(* IEC 61131-3 sources: B-R/Processes/EDT (part 2) *)

(* ---- EDTP2S3A_ACTION.st ---- *)
ACTION P2S3A_ACT:
	//设定时间
	FOR i := 0 TO EDTP2S3_STEP_NUM DO
		IF EDTP2S3A_ST[i] < T#5s THEN
			EDTP2S3A_ST[i] := T#5s;
		END_IF;
		EDTP2S3A_STEP[i].set_time := EDTP2S3A_ST[i];
	END_FOR;

	//流程步骤
	ProcessHandleFC(EDTP2S3A,EDTP2S3A_STEP[0],EDTP2S3_STEP_NUM);

	//object 手自动切换
	IF (EDTP2S3A.status.mode <> 0) AND (NOT EDTP2S3A.auto_mode_edge) THEN
		EDTP2S3A.auto_mode_edge := TRUE;
		EDTP2S3A.manual_mode_edge := FALSE;

		EDTTV0601E.control.auto_operate := TRUE;
		EDTTV0601D.control.auto_operate := TRUE;
		EDTTV0601F.control.auto_operate := TRUE;
		EDTXV0641.control.auto_operate := TRUE;
		EDTR05A.control.auto_operate := TRUE;
	END_IF;

	IF (EDTP2S3A.status.mode = 0) AND (NOT EDTP2S3A.manual_mode_edge) THEN
		EDTP2S3A.manual_mode_edge := TRUE;
		EDTP2S3A.auto_mode_edge := FALSE;

		EDTTV0601E.control.manual_operate := TRUE;
		EDTTV0601D.control.manual_operate := TRUE;
		EDTTV0601F.control.manual_operate := TRUE;
		EDTXV0641.control.manual_operate := TRUE;
		EDTR05A.control.manual_operate := TRUE;
	END_IF;

	//错误信号停机
	EDTP2S3A.input.error_signal := (EDTTV0601E.status.valve_status >= 2) OR (EDTR05A.status.motor_status >= 2) OR
	(EDTTV0601D.status.valve_status >= 2) OR (EDTTV0601F.status.valve_status >= 2) OR (EDTXV0641.status.valve_status >= 2);

	IF EDTP2S3A.status.run_state = 1 THEN
		//步骤执行动作
		CASE EDTP2S3A.status.run_step OF
			0:
				//初始化
				IF NOT EDTP2S3A_STEP[0].done THEN
					EDTTV0601E.control.auto_operate := TRUE;
					EDTTV0601D.control.auto_operate := TRUE;
					EDTTV0601F.control.auto_operate := TRUE;
					EDTXV0641.control.auto_operate := TRUE;
					EDTR05A.control.auto_operate := TRUE;
					EDTP2S3A_STEP[0].done := TRUE;
				END_IF;
			1:
				//人工投料
			2:
				CASE p2_step3_2a OF
					0:
						IF NOT EDTP2S3A_STEP[2].done THEN
							p2_step3_2a := 1;
						END_IF;
					1:
						EDTTV0601F.input.auto_open_signal := TRUE;
						IF EDTTV0601F.input.open_feedback_state THEN
							EDTXV0641.input.auto_open_signal := TRUE;
							p2_step3_2a := 2;
						END_IF;
					2:
						TON_38.PT := DINT_TO_TIME(EDTP2S3_PARA_T1 * 1000);
						TON_38.IN := TRUE;
						IF TON_38.Q THEN
							TON_38.IN := FALSE;
							p2_step3_2a := 3;
						END_IF;
					3:
						EDTTV0601F.input.auto_open_signal := FALSE;
						EDTXV0641.input.auto_open_signal := FALSE;
						IF EDTTV0601F.input.close_feedback_state THEN
							p2_step3_2a := 4;
						END_IF;
					4:
						EDTTV0601E.input.auto_open_signal := TRUE;
						IF EDTTV0601E.input.open_feedback_state THEN
							EDTTV0601D.input.auto_open_signal := TRUE;
							IF EDTTV0601D.input.open_feedback_state THEN
								p2_step3_2a := 5;
							END_IF;
						END_IF;
					5:
						IF EDTTIT0601.status.value >= EDTP2S3_PARA_Temp1 THEN
							p2_step3_2a := 0;
							EDTP2S3A_STEP[2].done := TRUE;
						END_IF;
				END_CASE;
				TON_38();
			3:
				//人工确认釜内回收情况
			4:
				EDTTV0601D.input.auto_open_signal := FALSE;
				IF EDTTV0601D.input.close_feedback_state THEN
					EDTTV0601E.input.auto_open_signal := FALSE;
					IF EDTTV0601E.input.close_feedback_state THEN
						EDTTV0601F.input.auto_open_signal := TRUE;
						IF EDTTV0601F.input.open_feedback_state THEN
							EDTP2S3A_STEP[4].done := TRUE;
						END_IF;
					END_IF;
				END_IF;
			5:
				//人工加料
			6:
				CASE p2_step3_6a OF
					0:
						IF NOT EDTP2S3A_STEP[6].done THEN
							p2_step3_6a := 1;
						END_IF;
					1:
						EDTTV0601F.input.auto_open_signal := TRUE;
						IF EDTTV0601F.input.open_feedback_state THEN
							EDTXV0641.input.auto_open_signal := TRUE;
							p2_step3_6a := 2;
						END_IF;
					2:
						TON_39.PT := DINT_TO_TIME(EDTP2S3_PARA_T1 * 1000);
						TON_39.IN := TRUE;
						IF TON_39.Q THEN
							TON_39.IN := FALSE;
							p2_step3_6a := 3;
						END_IF;
					3:
						EDTTV0601F.input.auto_open_signal := FALSE;
						EDTXV0641.input.auto_open_signal := FALSE;
						IF EDTTV0601F.input.close_feedback_state THEN
							p2_step3_6a := 4;
						END_IF;
					4:
						EDTTV0601E.input.auto_open_signal := TRUE;
						IF EDTTV0601E.input.open_feedback_state THEN
							EDTTV0601D.input.auto_open_signal := TRUE;
							IF EDTTV0601D.input.open_feedback_state THEN
								p2_step3_6a := 5;
							END_IF;
						END_IF;
					5:
						IF EDTTIT0601.status.value >= EDTP2S3_PARA_Temp2 THEN
							p2_step3_6a := 0;
							EDTP2S3A_STEP[6].done := TRUE;
						END_IF;
				END_CASE;
				TON_39();
			7:
				//观察釜内情况
			8:
				EDTTV0601D.input.auto_open_signal := FALSE;
				IF EDTTV0601D.input.close_feedback_state THEN
					EDTTV0601E.input.auto_open_signal := FALSE;
					IF EDTTV0601E.input.close_feedback_state THEN
						EDTTV0601F.input.auto_open_signal := TRUE;
						IF EDTTV0601F.input.open_feedback_state THEN
							EDTP2S3A_STEP[8].done := TRUE;
						END_IF;
					END_IF;
				END_IF;
			9:
				//人工进料
			10:
				TON_10.PT := DINT_TO_TIME(EDTP2S3_PARA_T2 * 60 * 1000);
				TON_10.IN := TRUE;
				IF TON_10.Q THEN
					TON_10.IN := FALSE;
					EDTR05A.input.auto_run_signal := FALSE;
					EDTP2S3A_STEP[10].done := TRUE;
				END_IF;
				TON_10();
		END_CASE;
	END_IF;

	//人工确认步骤可用
	IF (EDTP2S3A.status.run_state) AND (NOT EDTP2S3A_STEP[EDTP2S3A.status.run_step].done AND ((EDTP2S3A.status.run_step = 1) OR (EDTP2S3A.status.run_step = 3) OR (EDTP2S3A.status.run_step = 5) OR (EDTP2S3A.status.run_step = 7) OR
		(EDTP2S3A.status.run_step = 9))) THEN
		EDTP2S3A.status.confirm_enable := TRUE;
	ELSE
		EDTP2S3A.status.confirm_enable := FALSE;
	END_IF;

END_ACTION

(* ---- EDTP2S3B_ACTION.st ---- *)
ACTION P2S3B_ACT:
	//设定时间
	FOR i := 0 TO EDTP2S3_STEP_NUM DO
		IF EDTP2S3B_ST[i] < T#5s THEN
			EDTP2S3B_ST[i] := T#5s;
		END_IF;
		EDTP2S3B_STEP[i].set_time := EDTP2S3B_ST[i];
	END_FOR;

	//流程步骤
	ProcessHandleFC(EDTP2S3B,EDTP2S3B_STEP[0],EDTP2S3_STEP_NUM);

	//object 手自动切换
	IF (EDTP2S3B.status.mode <> 0) AND (NOT EDTP2S3B.auto_mode_edge) THEN
		EDTP2S3B.auto_mode_edge := TRUE;
		EDTP2S3B.manual_mode_edge := FALSE;

		EDTTV0603E.control.auto_operate := TRUE;
		EDTTV0603D.control.auto_operate := TRUE;
		EDTTV0603F.control.auto_operate := TRUE;
		EDTXV0642.control.auto_operate := TRUE;
		EDTR05B.control.auto_operate := TRUE;
	END_IF;

	IF (EDTP2S3B.status.mode = 0) AND (NOT EDTP2S3B.manual_mode_edge) THEN
		EDTP2S3B.manual_mode_edge := TRUE;
		EDTP2S3B.auto_mode_edge := FALSE;

		EDTTV0603E.control.manual_operate := TRUE;
		EDTTV0603D.control.manual_operate := TRUE;
		EDTTV0603F.control.manual_operate := TRUE;
		EDTXV0642.control.manual_operate := TRUE;
		EDTR05B.control.manual_operate := TRUE;
	END_IF;

	//错误信号停机
	EDTP2S3B.input.error_signal := (EDTTV0603E.status.valve_status >= 2) OR (EDTR05B.status.motor_status >= 2) OR
	(EDTTV0603D.status.valve_status >= 2) OR (EDTTV0603F.status.valve_status >= 2) OR (EDTXV0642.status.valve_status >= 2);

	IF EDTP2S3B.status.run_state = 1 THEN
		//步骤执行动作
		CASE EDTP2S3B.status.run_step OF
			0:
				//初始化
				IF NOT EDTP2S3B_STEP[0].done THEN
					EDTTV0603E.control.auto_operate := TRUE;
					EDTTV0603D.control.auto_operate := TRUE;
					EDTTV0603F.control.auto_operate := TRUE;
					EDTXV0642.control.auto_operate := TRUE;
					EDTR05B.control.auto_operate := TRUE;
					EDTP2S3B_STEP[0].done := TRUE;
				END_IF;
			1:
				//人工投料
			2:
				CASE p2_step3_2b OF
					0:
						IF NOT EDTP2S3B_STEP[2].done THEN
							p2_step3_2b := 1;
						END_IF;
					1:
						EDTTV0603F.input.auto_open_signal := TRUE;
						IF EDTTV0603F.input.open_feedback_state THEN
							EDTXV0642.input.auto_open_signal := TRUE;
							p2_step3_2b := 2;
						END_IF;
					2:
						TON_44.PT := DINT_TO_TIME(EDTP2S3_PARA_T1 * 1000);
						TON_44.IN := TRUE;
						IF TON_44.Q THEN
							TON_44.IN := FALSE;
							p2_step3_2b := 3;
						END_IF;
					3:
						EDTTV0603F.input.auto_open_signal := FALSE;
						EDTXV0642.input.auto_open_signal := FALSE;
						IF EDTTV0603F.input.close_feedback_state THEN
							p2_step3_2b := 4;
						END_IF;
					4:
						EDTTV0603E.input.auto_open_signal := TRUE;
						IF EDTTV0603E.input.open_feedback_state THEN
							EDTTV0603D.input.auto_open_signal := TRUE;
							IF EDTTV0603D.input.open_feedback_state THEN
								p2_step3_2b := 5;
							END_IF;
						END_IF;
					5:
						IF EDTTIT0603.status.value >= EDTP2S3_PARA_Temp1 THEN
							p2_step3_2b := 0;
							EDTP2S3B_STEP[2].done := TRUE;
						END_IF;
				END_CASE;
				TON_44();
			3:
				//人工确认釜内回收情况
			4:
				EDTTV0603D.input.auto_open_signal := FALSE;
				IF EDTTV0603D.input.close_feedback_state THEN
					EDTTV0603E.input.auto_open_signal := FALSE;
					IF EDTTV0603E.input.close_feedback_state THEN
						EDTTV0603F.input.auto_open_signal := TRUE;
						IF EDTTV0603F.input.open_feedback_state THEN
							EDTP2S3B_STEP[4].done := TRUE;
						END_IF;
					END_IF;
				END_IF;
			5:
				//人工加料
			6:
				CASE p2_step3_6b OF
					0:
						IF NOT EDTP2S3B_STEP[6].done THEN
							p2_step3_6b := 1;
						END_IF;
					1:
						EDTTV0603F.input.auto_open_signal := TRUE;
						IF EDTTV0603F.input.open_feedback_state THEN
							EDTXV0642.input.auto_open_signal := TRUE;
							p2_step3_6b := 2;
						END_IF;
					2:
						TON_47.PT := DINT_TO_TIME(EDTP2S3_PARA_T1 * 1000);
						TON_47.IN := TRUE;
						IF TON_47.Q THEN
							TON_47.IN := FALSE;
							p2_step3_6b := 3;
						END_IF;
					3:
						EDTTV0603F.input.auto_open_signal := FALSE;
						EDTXV0642.input.auto_open_signal := FALSE;
						IF EDTTV0603F.input.close_feedback_state THEN
							p2_step3_6b := 4;
						END_IF;
					4:
						EDTTV0603E.input.auto_open_signal := TRUE;
						IF EDTTV0603E.input.open_feedback_state THEN
							EDTTV0603D.input.auto_open_signal := TRUE;
							IF EDTTV0603D.input.open_feedback_state THEN
								p2_step3_6b := 5;
							END_IF;
						END_IF;
					5:
						IF EDTTIT0603.status.value >= EDTP2S3_PARA_Temp2 THEN
							p2_step3_6b := 0;
							EDTP2S3B_STEP[6].done := TRUE;
						END_IF;
				END_CASE;
				TON_47();
			7:
				//观察釜内情况
			8:
				EDTTV0603D.input.auto_open_signal := FALSE;
				IF EDTTV0603D.input.close_feedback_state THEN
					EDTTV0603E.input.auto_open_signal := FALSE;
					IF EDTTV0603E.input.close_feedback_state THEN
						EDTTV0603F.input.auto_open_signal := TRUE;
						IF EDTTV0603F.input.open_feedback_state THEN
							EDTP2S3B_STEP[8].done := TRUE;
						END_IF;
					END_IF;
				END_IF;
			9:
				//人工进料
			10:
				TON_48.PT := DINT_TO_TIME(EDTP2S3_PARA_T2 * 60 * 1000);
				TON_48.IN := TRUE;
				IF TON_48.Q THEN
					TON_48.IN := FALSE;
					EDTR05B.input.auto_run_signal := FALSE;
					EDTP2S3B_STEP[10].done := TRUE;
				END_IF;
				TON_48();
		END_CASE;
	END_IF;

	//人工确认步骤可用
	IF (EDTP2S3B.status.run_state) AND (NOT EDTP2S3B_STEP[EDTP2S3B.status.run_step].done AND ((EDTP2S3B.status.run_step = 1) OR (EDTP2S3B.status.run_step = 3) OR (EDTP2S3B.status.run_step = 5) OR (EDTP2S3B.status.run_step = 7) OR
		(EDTP2S3B.status.run_step = 9))) THEN
		EDTP2S3B.status.confirm_enable := TRUE;
	ELSE
		EDTP2S3B.status.confirm_enable := FALSE;
	END_IF;

END_ACTION

(* ---- EDTP2S3C_ACTION.st ---- *)
ACTION P2S3C_ACT:
	//设定时间
	FOR i := 0 TO EDTP2S3_STEP_NUM DO
		IF EDTP2S3C_ST[i] < T#5s THEN
			EDTP2S3C_ST[i] := T#5s;
		END_IF;
		EDTP2S3C_STEP[i].set_time := EDTP2S3C_ST[i];
	END_FOR;

	//流程步骤
	ProcessHandleFC(EDTP2S3C,EDTP2S3C_STEP[0],EDTP2S3_STEP_NUM);

	//object 手自动切换
	IF (EDTP2S3C.status.mode <> 0) AND (NOT EDTP2S3C.auto_mode_edge) THEN
		EDTP2S3C.auto_mode_edge := TRUE;
		EDTP2S3C.manual_mode_edge := FALSE;

		EDTTV0605E.control.auto_operate := TRUE;
		EDTTV0605D.control.auto_operate := TRUE;
		EDTTV0605F.control.auto_operate := TRUE;
		EDTXV0643.control.auto_operate := TRUE;
		EDTR05C.control.auto_operate := TRUE;
	END_IF;

	IF (EDTP2S3C.status.mode = 0) AND (NOT EDTP2S3C.manual_mode_edge) THEN
		EDTP2S3C.manual_mode_edge := TRUE;
		EDTP2S3C.auto_mode_edge := FALSE;

		EDTTV0605E.control.manual_operate := TRUE;
		EDTTV0605D.control.manual_operate := TRUE;
		EDTTV0605F.control.manual_operate := TRUE;
		EDTXV0643.control.manual_operate := TRUE;
		EDTR05C.control.manual_operate := TRUE;
	END_IF;

	//错误信号停机
	EDTP2S3C.input.error_signal := (EDTTV0605E.status.valve_status >= 2) OR (EDTR05C.status.motor_status >= 2) OR
	(EDTTV0605D.status.valve_status >= 2) OR (EDTTV0605F.status.valve_status >= 2) OR (EDTXV0643.status.valve_status >= 2);

	IF EDTP2S3C.status.run_state = 1 THEN
		//步骤执行动作
		CASE EDTP2S3C.status.run_step OF
			0:
				//初始化
				IF NOT EDTP2S3C_STEP[0].done THEN
					EDTTV0605E.control.auto_operate := TRUE;
					EDTTV0605D.control.auto_operate := TRUE;
					EDTTV0605F.control.auto_operate := TRUE;
					EDTXV0643.control.auto_operate := TRUE;
					EDTR05C.control.auto_operate := TRUE;
					EDTP2S3C_STEP[0].done := TRUE;
				END_IF;
			1:
				//人工投料
			2:
				CASE p2_step3_2c OF
					0:
						IF NOT EDTP2S3C_STEP[2].done THEN
							p2_step3_2c := 1;
						END_IF;
					1:
						EDTTV0605F.input.auto_open_signal := TRUE;
						IF EDTTV0605F.input.open_feedback_state THEN
							EDTXV0643.input.auto_open_signal := TRUE;
							p2_step3_2c := 2;
						END_IF;
					2:
						TON_50.PT := DINT_TO_TIME(EDTP2S3_PARA_T1 * 1000);
						TON_50.IN := TRUE;
						IF TON_50.Q THEN
							TON_50.IN := FALSE;
							p2_step3_2c := 3;
						END_IF;
					3:
						EDTTV0605F.input.auto_open_signal := FALSE;
						EDTXV0643.input.auto_open_signal := FALSE;
						IF EDTTV0605F.input.close_feedback_state THEN
							p2_step3_2c := 4;
						END_IF;
					4:
						EDTTV0605E.input.auto_open_signal := TRUE;
						IF EDTTV0605E.input.open_feedback_state THEN
							EDTTV0605D.input.auto_open_signal := TRUE;
							IF EDTTV0605D.input.open_feedback_state THEN
								p2_step3_2c := 5;
							END_IF;
						END_IF;
					5:
						IF EDTTIT0605.status.value >= EDTP2S3_PARA_Temp1 THEN
							p2_step3_2c := 0;
							EDTP2S3C_STEP[2].done := TRUE;
						END_IF;
				END_CASE;
				TON_50();
			3:
				//人工确认釜内回收情况
			4:
				EDTTV0605D.input.auto_open_signal := FALSE;
				IF EDTTV0605D.input.close_feedback_state THEN
					EDTTV0605E.input.auto_open_signal := FALSE;
					IF EDTTV0605E.input.close_feedback_state THEN
						EDTTV0605F.input.auto_open_signal := TRUE;
						IF EDTTV0605F.input.open_feedback_state THEN
							EDTP2S3C_STEP[4].done := TRUE;
						END_IF;
					END_IF;
				END_IF;
			5:
				//人工加料
			6:
				CASE p2_step3_6c OF
					0:
						IF NOT EDTP2S3C_STEP[6].done THEN
							p2_step3_6c := 1;
						END_IF;
					1:
						EDTTV0605F.input.auto_open_signal := TRUE;
						IF EDTTV0605F.input.open_feedback_state THEN
							EDTXV0643.input.auto_open_signal := TRUE;
							p2_step3_6c := 2;
						END_IF;
					2:
						TON_51.PT := DINT_TO_TIME(EDTP2S3_PARA_T1 * 1000);
						TON_51.IN := TRUE;
						IF TON_51.Q THEN
							TON_51.IN := FALSE;
							p2_step3_6c := 3;
						END_IF;
					3:
						EDTTV0605F.input.auto_open_signal := FALSE;
						EDTXV0643.input.auto_open_signal := FALSE;
						IF EDTTV0605F.input.close_feedback_state THEN
							p2_step3_6c := 4;
						END_IF;
					4:
						EDTTV0605E.input.auto_open_signal := TRUE;
						IF EDTTV0605E.input.open_feedback_state THEN
							EDTTV0605D.input.auto_open_signal := TRUE;
							IF EDTTV0605D.input.open_feedback_state THEN
								p2_step3_6c := 5;
							END_IF;
						END_IF;
					5:
						IF EDTTIT0605.status.value >= EDTP2S3_PARA_Temp2 THEN
							p2_step3_6c := 0;
							EDTP2S3C_STEP[6].done := TRUE;
						END_IF;
				END_CASE;
				TON_51();
			7:
				//观察釜内情况
			8:
				EDTTV0605D.input.auto_open_signal := FALSE;
				IF EDTTV0605D.input.close_feedback_state THEN
					EDTTV0605E.input.auto_open_signal := FALSE;
					IF EDTTV0605E.input.close_feedback_state THEN
						EDTTV0605F.input.auto_open_signal := TRUE;
						IF EDTTV0605F.input.open_feedback_state THEN
							EDTP2S3C_STEP[8].done := TRUE;
						END_IF;
					END_IF;
				END_IF;
			9:
				//人工进料
			10:
				TON_53.PT := DINT_TO_TIME(EDTP2S3_PARA_T2 * 60 * 1000);
				TON_53.IN := TRUE;
				IF TON_53.Q THEN
					TON_53.IN := FALSE;
					EDTR05C.input.auto_run_signal := FALSE;
					EDTP2S3C_STEP[10].done := TRUE;
				END_IF;
				TON_53();
		END_CASE;
	END_IF;

	//人工确认步骤可用
	IF (EDTP2S3C.status.run_state) AND (NOT EDTP2S3C_STEP[EDTP2S3C.status.run_step].done AND ((EDTP2S3C.status.run_step = 1) OR (EDTP2S3C.status.run_step = 3) OR (EDTP2S3C.status.run_step = 5) OR (EDTP2S3C.status.run_step = 7) OR
		(EDTP2S3C.status.run_step = 9))) THEN
		EDTP2S3C.status.confirm_enable := TRUE;
	ELSE
		EDTP2S3C.status.confirm_enable := FALSE;
	END_IF;

END_ACTION

(* ---- EDTP2S3D_ACTION.st ---- *)
ACTION P2S3D_ACT:
	//设定时间
	FOR i := 0 TO EDTP2S3_STEP_NUM DO
		IF EDTP2S3D_ST[i] < T#5s THEN
			EDTP2S3D_ST[i] := T#5s;
		END_IF;
		EDTP2S3D_STEP[i].set_time := EDTP2S3D_ST[i];
	END_FOR;

	//流程步骤
	ProcessHandleFC(EDTP2S3D,EDTP2S3D_STEP[0],EDTP2S3_STEP_NUM);

	//object 手自动切换
	IF (EDTP2S3D.status.mode <> 0) AND (NOT EDTP2S3D.auto_mode_edge) THEN
		EDTP2S3D.auto_mode_edge := TRUE;
		EDTP2S3D.manual_mode_edge := FALSE;

		EDTTV0607E.control.auto_operate := TRUE;
		EDTTV0607D.control.auto_operate := TRUE;
		EDTTV0607F.control.auto_operate := TRUE;
		EDTXV0644.control.auto_operate := TRUE;
		EDTR05D.control.auto_operate := TRUE;
	END_IF;

	IF (EDTP2S3D.status.mode = 0) AND (NOT EDTP2S3D.manual_mode_edge) THEN
		EDTP2S3D.manual_mode_edge := TRUE;
		EDTP2S3D.auto_mode_edge := FALSE;

		EDTTV0607E.control.manual_operate := TRUE;
		EDTTV0607D.control.manual_operate := TRUE;
		EDTTV0607F.control.manual_operate := TRUE;
		EDTXV0644.control.manual_operate := TRUE;
		EDTR05D.control.manual_operate := TRUE;
	END_IF;

	//错误信号停机
	EDTP2S3D.input.error_signal := (EDTTV0607E.status.valve_status >= 2) OR (EDTR05D.status.motor_status >= 2) OR
	(EDTTV0607D.status.valve_status >= 2) OR (EDTTV0607F.status.valve_status >= 2) OR (EDTXV0644.status.valve_status >= 2);

	IF EDTP2S3D.status.run_state = 1 THEN
		//步骤执行动作
		CASE EDTP2S3D.status.run_step OF
			0:
				//初始化
				IF NOT EDTP2S3D_STEP[0].done THEN
					EDTTV0607E.control.auto_operate := TRUE;
					EDTTV0607D.control.auto_operate := TRUE;
					EDTTV0607F.control.auto_operate := TRUE;
					EDTXV0644.control.auto_operate := TRUE;
					EDTR05D.control.auto_operate := TRUE;
					EDTP2S3D_STEP[0].done := TRUE;
				END_IF;
			1:
				//人工投料
			2:
				CASE p2_step3_2d OF
					0:
						IF NOT EDTP2S3D_STEP[2].done THEN
							p2_step3_2d := 1;
						END_IF;
					1:
						EDTTV0607F.input.auto_open_signal := TRUE;
						IF EDTTV0607F.input.open_feedback_state THEN
							EDTXV0644.input.auto_open_signal := TRUE;
							p2_step3_2d := 2;
						END_IF;
					2:
						TON_56.PT := DINT_TO_TIME(EDTP2S3_PARA_T1 * 1000);
						TON_56.IN := TRUE;
						IF TON_56.Q THEN
							TON_56.IN := FALSE;
							p2_step3_2d := 3;
						END_IF;
					3:
						EDTTV0607F.input.auto_open_signal := FALSE;
						EDTXV0644.input.auto_open_signal := FALSE;
						IF EDTTV0607F.input.close_feedback_state THEN
							p2_step3_2d := 4;
						END_IF;
					4:
						EDTTV0607E.input.auto_open_signal := TRUE;
						IF EDTTV0607E.input.open_feedback_state THEN
							EDTTV0607D.input.auto_open_signal := TRUE;
							IF EDTTV0607D.input.open_feedback_state THEN
								p2_step3_2d := 5;
							END_IF;
						END_IF;
					5:
						IF EDTTIT0607.status.value >= EDTP2S3_PARA_Temp1 THEN
							p2_step3_2d := 0;
							EDTP2S3D_STEP[2].done := TRUE;
						END_IF;
				END_CASE;
				TON_56();
			3:
				//人工确认釜内回收情况
			4:
				EDTTV0607D.input.auto_open_signal := FALSE;
				IF EDTTV0607D.input.close_feedback_state THEN
					EDTTV0607E.input.auto_open_signal := FALSE;
					IF EDTTV0607E.input.close_feedback_state THEN
						EDTTV0607F.input.auto_open_signal := TRUE;
						IF EDTTV0607F.input.open_feedback_state THEN
							EDTP2S3D_STEP[4].done := TRUE;
						END_IF;
					END_IF;
				END_IF;
			5:
				//人工加料
			6:
				CASE p2_step3_6d OF
					0:
						IF NOT EDTP2S3D_STEP[6].done THEN
							p2_step3_6d := 1;
						END_IF;
					1:
						EDTTV0607F.input.auto_open_signal := TRUE;
						IF EDTTV0607F.input.open_feedback_state THEN
							EDTXV0644.input.auto_open_signal := TRUE;
							p2_step3_6d := 2;
						END_IF;
					2:
						TON_57.PT := DINT_TO_TIME(EDTP2S3_PARA_T1 * 1000);
						TON_57.IN := TRUE;
						IF TON_57.Q THEN
							TON_57.IN := FALSE;
							p2_step3_6d := 3;
						END_IF;
					3:
						EDTTV0607F.input.auto_open_signal := FALSE;
						EDTXV0644.input.auto_open_signal := FALSE;
						IF EDTTV0607F.input.close_feedback_state THEN
							p2_step3_6d := 4;
						END_IF;
					4:
						EDTTV0607E.input.auto_open_signal := TRUE;
						IF EDTTV0607E.input.open_feedback_state THEN
							EDTTV0607D.input.auto_open_signal := TRUE;
							IF EDTTV0607D.input.open_feedback_state THEN
								p2_step3_6d := 5;
							END_IF;
						END_IF;
					5:
						IF EDTTIT0607.status.value >= EDTP2S3_PARA_Temp2 THEN
							p2_step3_6d := 0;
							EDTP2S3D_STEP[6].done := TRUE;
						END_IF;
				END_CASE;
				TON_57();
			7:
				//观察釜内情况
			8:
				EDTTV0607D.input.auto_open_signal := FALSE;
				IF EDTTV0607D.input.close_feedback_state THEN
					EDTTV0607E.input.auto_open_signal := FALSE;
					IF EDTTV0607E.input.close_feedback_state THEN
						EDTTV0607F.input.auto_open_signal := TRUE;
						IF EDTTV0607F.input.open_feedback_state THEN
							EDTP2S3D_STEP[8].done := TRUE;
						END_IF;
					END_IF;
				END_IF;
			9:
				//人工进料
			10:
				TON_59.PT := DINT_TO_TIME(EDTP2S3_PARA_T2 * 60 * 1000);
				TON_59.IN := TRUE;
				IF TON_59.Q THEN
					TON_59.IN := FALSE;
					EDTR05D.input.auto_run_signal := FALSE;
					EDTP2S3D_STEP[10].done := TRUE;
				END_IF;
				TON_59();
		END_CASE;
	END_IF;

	//人工确认步骤可用
	IF (EDTP2S3D.status.run_state) AND (NOT EDTP2S3D_STEP[EDTP2S3D.status.run_step].done AND ((EDTP2S3D.status.run_step = 1) OR (EDTP2S3D.status.run_step = 3) OR (EDTP2S3D.status.run_step = 5) OR (EDTP2S3D.status.run_step = 7) OR
		(EDTP2S3D.status.run_step = 9))) THEN
		EDTP2S3D.status.confirm_enable := TRUE;
	ELSE
		EDTP2S3D.status.confirm_enable := FALSE;
	END_IF;

END_ACTION

(* ---- EDTP2S4A_ACTION.st ---- *)
ACTION P2S4A_ACT:
	//设定时间
	FOR i := 0 TO EDTP2S4_STEP_NUM DO
		IF EDTP2S4A_ST[i] < T#5s THEN
			EDTP2S4A_ST[i] := T#5s;
		END_IF;
		EDTP2S4A_STEP[i].set_time := EDTP2S4A_ST[i];
	END_FOR;

	//流程步骤
	ProcessHandleFC(EDTP2S4A,EDTP2S4A_STEP[0],EDTP2S4_STEP_NUM);

	//object 手自动切换
	IF (EDTP2S4A.status.mode <> 0) AND (NOT EDTP2S4A.auto_mode_edge) THEN
		EDTP2S4A.auto_mode_edge := TRUE;
		EDTP2S4A.manual_mode_edge := FALSE;

		EDTXV0711.control.auto_operate := TRUE;
		EDTAV0701B.control.auto_operate := TRUE;
		EDTAV0701A.control.auto_operate := TRUE;
		EDTXV0701.control.auto_operate := TRUE;
		EDTR12A.control.auto_operate := TRUE;
		EDTTV0701C.control.auto_operate := TRUE;
		EDTTV0701D.control.auto_operate := TRUE;
		EDTTV0701E.control.auto_operate := TRUE;
		EDTTV0701F.control.auto_operate := TRUE;
		EDTFVT0701.control.auto_operate := TRUE;
		EDTXV0704.control.auto_operate := TRUE;
		EDTXV0705.control.auto_operate := TRUE;
		EDTTV0701A.control.auto_operate := TRUE;
		EDTTV0701B.control.auto_operate := TRUE;
		EDTXV0708.control.auto_operate := TRUE;
		EDTXV0709.control.auto_operate := TRUE;
		EDTXV0715.control.auto_operate := TRUE;

	END_IF;

	IF (EDTP2S4A.status.mode = 0) AND (NOT EDTP2S4A.manual_mode_edge) THEN
		EDTP2S4A.manual_mode_edge := TRUE;
		EDTP2S4A.auto_mode_edge := FALSE;

		EDTXV0711.control.manual_operate := TRUE;
		EDTAV0701B.control.manual_operate := TRUE;
		EDTAV0701A.control.manual_operate := TRUE;
		EDTXV0701.control.manual_operate := TRUE;
		EDTR12A.control.manual_operate := TRUE;
		EDTTV0701C.control.manual_operate := TRUE;
		EDTTV0701D.control.manual_operate := TRUE;
		EDTTV0701E.control.manual_operate := TRUE;
		EDTTV0701F.control.manual_operate := TRUE;
		EDTFVT0701.control.manual_operate := TRUE;
		EDTXV0704.control.manual_operate := TRUE;
		EDTXV0705.control.manual_operate := TRUE;
		EDTTV0701A.control.manual_operate := TRUE;
		EDTTV0701B.control.manual_operate := TRUE;
		EDTXV0708.control.manual_operate := TRUE;
		EDTXV0709.control.manual_operate := TRUE;
		EDTXV0715.control.manual_operate := TRUE;
	END_IF;

	//错误信号停机
	EDTP2S4A.input.error_signal := (EDTXV0711.status.valve_status >= 2) OR (EDTAV0701B.status.valve_status >= 2) OR
	(EDTR12A.status.motor_status >= 2) OR (EDTAV0701A.status.valve_status >= 2) OR (EDTXV0701.status.valve_status >= 2) OR
	(EDTTV0701C.status.valve_status >= 2) OR (EDTTV0701D.status.valve_status >= 2) OR (EDTTV0701E.status.valve_status >= 2) OR
	(EDTTV0701F.status.valve_status >= 2) OR (EDTXV0704.status.valve_status >= 2) OR (EDTXV0705.status.valve_status >= 2) OR
	(EDTTV0701A.status.valve_status >= 2) OR (EDTTV0701B.status.valve_status >= 2) OR (EDTXV0708.status.valve_status >= 2) OR
	(EDTXV0709.status.valve_status >= 2);

	IF EDTP2S4A.status.run_state = 1 THEN
		//步骤执行动作
		CASE EDTP2S4A.status.run_step OF
			0:
				//初始化
				IF NOT EDTP2S4A_STEP[0].done THEN
					EDTXV0711.control.auto_operate := TRUE;
					EDTAV0701B.control.auto_operate := TRUE;
					EDTAV0701A.control.auto_operate := TRUE;
					EDTXV0701.control.auto_operate := TRUE;
					EDTR12A.control.auto_operate := TRUE;
					EDTTV0701C.control.auto_operate := TRUE;
					EDTTV0701D.control.auto_operate := TRUE;
					EDTTV0701E.control.auto_operate := TRUE;
					EDTTV0701F.control.auto_operate := TRUE;
					EDTFVT0701.control.auto_operate := TRUE;
					EDTXV0704.control.auto_operate := TRUE;
					EDTXV0705.control.auto_operate := TRUE;
					EDTTV0701A.control.auto_operate := TRUE;
					EDTTV0701B.control.auto_operate := TRUE;
					EDTXV0708.control.auto_operate := TRUE;
					EDTXV0709.control.auto_operate := TRUE;
					EDTXV0715.control.auto_operate := TRUE;
					EDTP2S4A_STEP[0].done := TRUE;
				END_IF;
			1:
				//手动分层，完成后点确认
			2:
				//除前馏
				R12A_process1 := TRUE;
				EDTP2S4A_STEP[2].done := TRUE;
			3:
				IF NOT R12A_process1 THEN
					EDTP2S4A_STEP[3].done := TRUE;
				END_IF;
			4:
				//转移确认V19空
			5:
				TON_66.PT := DINT_TO_TIME(EDTP2S4_PARA_T5 * 60 * 1000);
				EDTXV0708.input.auto_open_signal := TRUE;
				IF EDTXV0708.input.open_feedback_state THEN
					TON_66.IN := TRUE;
				END_IF;
				IF TON_66.Q THEN
					TON_66.IN := FALSE;
					EDTP2S4A_STEP[5].done := TRUE;
				END_IF;
				TON_66();
			6:
				//确认R12A空
			7:
				TON_67.PT := DINT_TO_TIME(EDTP2S4_PARA_T6 * 60 * 1000);
				EDTXV0708.input.auto_open_signal := FALSE;
				IF EDTXV0708.input.close_feedback_state THEN
					EDTXV0711.input.auto_open_signal := TRUE;
					EDTAV0701A.input.auto_open_signal := TRUE;
				END_IF;
				IF EDTXV0711.input.open_feedback_state AND EDTAV0701A.input.open_feedback_state THEN
					TON_67.IN := TRUE;
				END_IF;
				IF TON_67.Q THEN
					TON_67.IN := FALSE;
					EDTP2S4A_STEP[7].done := TRUE;
				END_IF;
				TON_67();
			8:
				//确认R06A空
			9:
				R12A_process := TRUE;
				EDTAV0701A.input.auto_open_signal := FALSE;
				IF EDTAV0701A.input.close_feedback_state THEN
					EDTXV0711.input.auto_open_signal := FALSE;
					IF EDTXV0711.input.close_feedback_state THEN
						EDTXV0709.input.auto_open_signal := TRUE;
						IF EDTXV0709.input.open_feedback_state THEN
							EDTXV0715.input.auto_open_signal := TRUE;
							EDTP2S4A_STEP[9].done := TRUE;
						END_IF;
					END_IF;
				END_IF;
			10:
				//确认转移完毕，AV0701B前手阀开度为三分一
			11:
				EDTXV0709.input.auto_open_signal := FALSE;
				EDTXV0715.input.auto_open_signal := FALSE;
				EDTAV0701B.input.auto_open_signal := TRUE;
				EDTXV0711.input.auto_open_signal := TRUE;
				IF EDTXV0709.input.close_feedback_state AND EDTXV0711.input.open_feedback_state AND EDTAV0701B.input.open_feedback_state THEN
					EDTP2S4A_STEP[11].done := TRUE;
				END_IF;
			12:
				//V06-->V22确认转移完毕
			13:
				EDTAV0701B.input.auto_open_signal := FALSE;
				EDTXV0711.input.auto_open_signal := FALSE;
				IF EDTXV0711.input.close_feedback_state AND EDTAV0701B.input.close_feedback_state THEN
					EDTP2S4A_STEP[13].done := TRUE;
				END_IF;
			14:
				IF NOT R12A_process THEN
					EDTP2S4A_STEP[14].done := TRUE;
				END_IF;
			15:
			//转移
		END_CASE;
	END_IF;

	//除前馏
	IF R12A_process1 THEN
		CASE R12A_process1_step OF
			0:
				MTBasicsPID_8.Enable := FALSE;
				EDTXV0701.input.auto_open_signal := TRUE;
				EDTR12A.input.auto_run_signal := TRUE;
				EDTXV0704.input.auto_open_signal := FALSE;
				EDTXV0705.input.auto_open_signal := FALSE;
				EDTFVT0701.input.auto_degree_set := 0.0;
				IF EDTXV0701.input.open_feedback_state AND EDTR12A.input.run_feedback AND EDTXV0704.input.close_feedback_state AND EDTXV0705.input.close_feedback_state THEN
					R12A_process1_step := 1;
				END_IF;
			1:
				HeatPot_2(ST1 := DINT_TO_TIME(EDTP2S4_PARA_T2 * 1000),
				ST2 := DINT_TO_TIME(EDTP2S4_PARA_T3 * 1000),
				V3 := EDTTV0701C,
				V4 := EDTTV0701D,
				V5 := EDTTV0701E,
				V6 := EDTTV0701F,
				done := R12A_process1_step_1_done);
				IF R12A_process1_step_1_done THEN
					R12A_process1_step_1_done := FALSE;
					R12A_process1_step := 2;
				END_IF;
			2:
				IF EDTTIT0701.status.value >= EDTP2S4_PARA_Temp1 THEN
					EDTTV0701C.input.auto_open_signal := FALSE;
					IF EDTTV0701C.input.close_feedback_state THEN
						R12A_process1_step := 3;
					END_IF;
				END_IF;
			3:
				TON_24.PT := DINT_TO_TIME(EDTP2S4_PARA_T4 * 60 * 1000);
				IF EDTTIT0702.status.value >= EDTP2S4_PARA_Temp4 THEN
					TON_24.IN := TRUE;
				END_IF;
				IF TON_24.Q THEN
					TON_24.IN := FALSE;
					R12A_process1_step := 4;
				END_IF;
			4:
				MTBasicsPID_8.Enable := TRUE;
				EDTXV0705.input.auto_open_signal := FALSE;
				IF EDTXV0705.input.close_feedback_state THEN
					EDTXV0704.input.auto_open_signal := TRUE;
					IF EDTXV0704.input.open_feedback_state THEN
						//EDTFVT0701.input.auto_degree_set := EDTP2S4A_PARA_O1;
						R12A_process1_step := 5;
					END_IF;
				END_IF;
			5:
				TON_24.PT := DINT_TO_TIME(EDTP2S4_PARA_T7 * 1000);
				IF EDTTIT0702.status.value >= EDTP2S4_PARA_Temp2 THEN
					EDTTV0701D.input.auto_open_signal := FALSE;
					IF EDTTV0701D.input.close_feedback_state THEN
						EDTTV0701E.input.auto_open_signal := FALSE;
						EDTTV0701F.input.auto_open_signal := TRUE;
						//IF EDTTV0701E.input.close_feedback_state AND EDTTV0701F.input.open_feedback_state THEN
							TON_24.IN := TRUE;
						//END_IF;
					END_IF;
				END_IF;
				IF TON_24.Q THEN
					TON_24.IN := FALSE;
					R12A_process1_step := 6;
				END_IF;
			6:
				EDTTV0701F.input.auto_open_signal := FALSE;
				IF EDTTV0701F.input.close_feedback_state THEN
					EDTTV0701A.input.auto_open_signal := TRUE;
					IF EDTTV0701A.input.open_feedback_state THEN
						EDTTV0701B.input.auto_open_signal := TRUE;
						R12A_process1_step := 7;
					END_IF;
				END_IF;
			7:
				IF EDTTIT0701.status.value <= EDTP2S4_PARA_Temp3 THEN
					MTBasicsPID_8.Enable := FALSE;
					EDTTV0701B.input.auto_open_signal := FALSE;
					EDTTV0701A.input.auto_open_signal := FALSE;
					EDTR12A.input.auto_run_signal := FALSE;
					EDTXV0701.input.auto_open_signal := FALSE;
					EDTFVT0701.input.auto_degree_set := 100.0;
				END_IF;
				IF EDTTV0701A.input.close_feedback_state AND EDTTV0701B.input.close_feedback_state AND (NOT EDTR12A.input.run_feedback) THEN// AND EDTXV0701.input.close_feedback_state THEN
					R12A_process1 := FALSE;
					R12A_process1_step := 0;
				END_IF;
		END_CASE;
		TON_24();
	END_IF;

	//甲醇水蒸馏
	IF R12A_process THEN
		CASE R12A_process_step OF
			0:
				//甲醇水蒸馏准备
				MTBasicsPID_8.Enable := FALSE;
				EDTXV0704.input.auto_open_signal := FALSE;
				EDTXV0705.input.auto_open_signal := FALSE;
				EDTXV0701.input.auto_open_signal := TRUE;
				EDTR12A.input.auto_run_signal := TRUE;
				EDTFVT0701.input.auto_degree_set := 0.0;
				IF EDTXV0701.input.open_feedback_state AND EDTR12A.input.run_feedback AND EDTXV0704.input.close_feedback_state AND EDTXV0705.input.close_feedback_state THEN
					R12A_process_step := 1;
				END_IF;
			1:
				HeatPot_5(ST1 := DINT_TO_TIME(EDTP2S4_PARA_T2 * 1000),
				ST2 := DINT_TO_TIME(EDTP2S4_PARA_T3 * 1000),
				V3 := EDTTV0701C,
				V4 := EDTTV0701D,
				V5 := EDTTV0701E,
				V6 := EDTTV0701F,
				done := R12A_process_step_1_done);
				IF R12A_process_step_1_done THEN
					R12A_process_step_1_done := FALSE;
					R12A_process_step := 2;
				END_IF;
			2:
				IF EDTTIT0701.status.value >= EDTP2S4_PARA_Temp1 THEN
					EDTTV0701C.input.auto_open_signal := FALSE;
					IF EDTTV0701C.input.close_feedback_state THEN
						R12A_process_step := 3;
					END_IF;
				END_IF;
			3:
				TON_69.PT := DINT_TO_TIME(EDTP2S4_PARA_T4 * 60 * 1000);
				IF EDTTIT0702.status.value >= EDTP2S4_PARA_Temp4 THEN
					TON_69.IN := TRUE;
				END_IF;
				IF TON_69.Q THEN
					TON_69.IN := FALSE;
					R12A_process_step := 4;
				END_IF;
			4:
				MTBasicsPID_8.Enable := TRUE;
				EDTXV0705.input.auto_open_signal := FALSE;
				IF EDTXV0705.input.close_feedback_state THEN
					EDTXV0704.input.auto_open_signal := TRUE;
					IF EDTXV0704.input.open_feedback_state THEN
						//EDTFVT0701.input.auto_degree_set := EDTP2S4A_PARA_O2;
						R12A_process_step := 5;
					END_IF;
				END_IF;
			5:
				IF EDTTIT0702.status.value >= EDTP2S4_PARA_Temp5 THEN
					EDTXV0704.input.auto_open_signal := FALSE;
					IF EDTXV0704.input.close_feedback_state THEN
						EDTXV0705.input.auto_open_signal := TRUE;
						IF EDTXV0705.input.open_feedback_state THEN
							//EDTFVT0701.input.auto_degree_set := EDTP2S4A_PARA_O3;
							R12A_process_step := 6;
						END_IF;
					END_IF;
				END_IF;
			6:
				TON_69.PT := DINT_TO_TIME(EDTP2S4_PARA_T7 * 1000);
				IF EDTTIT0702.status.value >= EDTP2S4_PARA_Temp6 THEN
					EDTTV0701D.input.auto_open_signal := FALSE;
					IF EDTTV0701D.input.close_feedback_state THEN
						EDTTV0701E.input.auto_open_signal := FALSE;
						EDTTV0701F.input.auto_open_signal := TRUE;
						//IF EDTTV0701E.input.close_feedback_state AND EDTTV0701F.input.open_feedback_state THEN
							TON_69.IN := TRUE;
						//END_IF;
					END_IF;
				END_IF;
				IF TON_69.Q THEN
					TON_69.IN := FALSE;
					R12A_process_step := 7;
				END_IF;
			7:
				EDTTV0701F.input.auto_open_signal := FALSE;
				IF EDTTV0701F.input.close_feedback_state THEN
					EDTTV0701A.input.auto_open_signal := TRUE;
					IF EDTTV0701A.input.open_feedback_state THEN
						EDTTV0701B.input.auto_open_signal := TRUE;
						R12A_process_step := 8;
					END_IF;
				END_IF;
			8:
				IF EDTTIT0701.status.value <= EDTP2S4_PARA_Temp7 THEN
					MTBasicsPID_8.Enable := FALSE;
					EDTTV0701B.input.auto_open_signal := FALSE;
					EDTTV0701A.input.auto_open_signal := FALSE;
					EDTR12A.input.auto_run_signal := FALSE;
					EDTXV0701.input.auto_open_signal := FALSE;
					EDTFVT0701.input.auto_degree_set := 100.0;
				END_IF;
				IF EDTTV0701A.input.close_feedback_state AND EDTTV0701B.input.close_feedback_state AND (NOT EDTR12A.input.run_feedback) THEN //AND EDTXV0701.input.close_feedback_state THEN note：关反馈有问题 临时去掉
					R12A_process := FALSE;
					R12A_process_step := 0;
				END_IF;
		END_CASE;
		TON_69();
	END_IF;

	//分层
	IF r06a_separate THEN
		CASE r06a_separate_step OF
			0:
				r06a_als_data_last := r06a_als_data;
				EDTAV0701B.control.auto_operate := TRUE;
				r06a_separate_step := 1;
			1:
				TON_3.PT := T#2s;
				TON_3.IN := TRUE;
				IF TON_3.Q THEN
					TON_3.IN := FALSE;
					r06a_separate_step := 2;
				END_IF;
			2:
				IF r06a_als_data_last = r06a_als_data THEN
					r06a_separate := FALSE;
					r06a_separate_step := 0;
				ELSE
					r06a_separate_step := 3;
				END_IF;
			3:
				EDTAV0701B.input.auto_open_signal := TRUE;
				TON_3.PT := T#30s;
				TON_3.IN := TRUE;
				IF TON_3.Q THEN
					TON_3.IN := FALSE;
					r06a_separate_step := 4;
					r06a_als_data_last := r06a_als_data;
				END_IF;
			4:
				IF ABS(r06a_als_data_last - r06a_als_data) >= r06a_als_data_threshold THEN
					EDTAV0701B.input.auto_open_signal := FALSE;
					r06a_separate := FALSE;
					r06a_separate_step := 0;
				END_IF;
		END_CASE;
		TON_3();
	END_IF;

	R_TRIG_0(CLK := EDTFVT0701.status.auto_mode);
	IF R_TRIG_0.Q THEN
		MTBasicsPID_8.Enable := TRUE;
	END_IF;
	F_TRIG_0(CLK := EDTFVT0701.status.auto_mode);
	IF F_TRIG_0.Q THEN
		MTBasicsPID_8.Enable := FALSE;
	END_IF;
	//FVT0701 pid调节
	//	MTBasicsPID_8.Enable := TRUE;
	MTBasicsPID_8.PIDParameters.Gain := EDTPid0701Para.gain;
	MTBasicsPID_8.PIDParameters.IntegrationTime := EDTPid0701Para.integration_time;
	MTBasicsPID_8.PIDParameters.DerivativeTime := EDTPid0701Para.derivative_time;
	MTBasicsPID_8.MinOut := 0.0;
	MTBasicsPID_8.MaxOut := 100.0;
	MTBasicsPID_8.SetValue := EDTPid0701Para.set_value;
	MTBasicsPID_8.ActValue := EDTFIT0701.flowrate;
	MTBasicsPID_8.Update := EDTPid0701.update;
	MTBasicsPID_8();
	EDTPid0701.out := MTBasicsPID_8.Out;
	IF MTBasicsPID_8.Active THEN
		EDTFVT0701.input.auto_degree_set := MTBasicsPID_8.Out + EDTPid0701Para.min_out;
		//	ELSE
		//		EDTFVT0701.input.auto_degree_set := 0.0;
	END_IF;
	IF MTBasicsPID_8.UpdateDone THEN
		EDTPid0701.update := FALSE;
	END_IF;

	//人工确认步骤可用
	IF (EDTP2S4A.status.run_state) AND (NOT EDTP2S4A_STEP[EDTP2S4A.status.run_step].done AND ((EDTP2S4A.status.run_step = 1) OR (EDTP2S4A.status.run_step = 4)
		OR (EDTP2S4A.status.run_step = 6) OR (EDTP2S4A.status.run_step = 8) OR (EDTP2S4A.status.run_step = 10) OR (EDTP2S4A.status.run_step = 12) OR (EDTP2S4A.status.run_step = 15))) THEN
		EDTP2S4A.status.confirm_enable := TRUE;
	ELSE
		EDTP2S4A.status.confirm_enable := FALSE;
	END_IF;

END_ACTION

(* ---- EDTP2S4B_ACTION.st ---- *)
ACTION P2S4B_ACT:
	//设定时间
	FOR i := 0 TO EDTP2S4_STEP_NUM DO
		IF EDTP2S4B_ST[i] < T#5s THEN
			EDTP2S4B_ST[i] := T#5s;
		END_IF;
		EDTP2S4B_STEP[i].set_time := EDTP2S4B_ST[i];
	END_FOR;

	//流程步骤
	ProcessHandleFC(EDTP2S4B,EDTP2S4B_STEP[0],EDTP2S4_STEP_NUM);

	//object 手自动切换
	IF (EDTP2S4B.status.mode <> 0) AND (NOT EDTP2S4B.auto_mode_edge) THEN
		EDTP2S4B.auto_mode_edge := TRUE;
		EDTP2S4B.manual_mode_edge := FALSE;

		EDTXV0724.control.auto_operate := TRUE;
		EDTAV0702B.control.auto_operate := TRUE;
		EDTAV0702A.control.auto_operate := TRUE;
		EDTXV0716.control.auto_operate := TRUE;
		EDTR12B.control.auto_operate := TRUE;
		EDTTV0703C.control.auto_operate := TRUE;
		EDTTV0703D.control.auto_operate := TRUE;
		EDTTV0703E.control.auto_operate := TRUE;
		EDTTV0703F.control.auto_operate := TRUE;
		EDTFVT0703.control.auto_operate := TRUE;
		EDTXV0719.control.auto_operate := TRUE;
		EDTXV0718.control.auto_operate := TRUE;
		EDTTV0703A.control.auto_operate := TRUE;
		EDTTV0703B.control.auto_operate := TRUE;
		EDTXV0722.control.auto_operate := TRUE;
		EDTXV0723.control.auto_operate := TRUE;
		EDTXV0715.control.auto_operate := TRUE;

	END_IF;

	IF (EDTP2S4B.status.mode = 0) AND (NOT EDTP2S4B.manual_mode_edge) THEN
		EDTP2S4B.manual_mode_edge := TRUE;
		EDTP2S4B.auto_mode_edge := FALSE;

		EDTXV0724.control.manual_operate := TRUE;
		EDTAV0702B.control.manual_operate := TRUE;
		EDTAV0702A.control.manual_operate := TRUE;
		EDTXV0716.control.manual_operate := TRUE;
		EDTR12B.control.manual_operate := TRUE;
		EDTTV0703C.control.manual_operate := TRUE;
		EDTTV0703D.control.manual_operate := TRUE;
		EDTTV0703E.control.manual_operate := TRUE;
		EDTTV0703F.control.manual_operate := TRUE;
		EDTFVT0703.control.manual_operate := TRUE;
		EDTXV0719.control.manual_operate := TRUE;
		EDTXV0718.control.manual_operate := TRUE;
		EDTTV0703A.control.manual_operate := TRUE;
		EDTTV0703B.control.manual_operate := TRUE;
		EDTXV0722.control.manual_operate := TRUE;
		EDTXV0723.control.manual_operate := TRUE;
		EDTXV0715.control.manual_operate := TRUE;
	END_IF;

	//错误信号停机
	EDTP2S4B.input.error_signal := (EDTXV0724.status.valve_status >= 2) OR (EDTAV0702B.status.valve_status >= 2) OR
	(EDTR12B.status.motor_status >= 2) OR (EDTAV0702A.status.valve_status >= 2) OR (EDTXV0716.status.valve_status >= 2) OR
	(EDTTV0703C.status.valve_status >= 2) OR (EDTTV0703D.status.valve_status >= 2) OR (EDTTV0703E.status.valve_status >= 2) OR
	(EDTTV0703F.status.valve_status >= 2) OR (EDTXV0719.status.valve_status >= 2) OR (EDTXV0718.status.valve_status >= 2) OR
	(EDTTV0703A.status.valve_status >= 2) OR (EDTTV0703B.status.valve_status >= 2) OR (EDTXV0722.status.valve_status >= 2) OR
	(EDTXV0723.status.valve_status >= 2);

	IF EDTP2S4B.status.run_state = 1 THEN
		//步骤执行动作
		CASE EDTP2S4B.status.run_step OF
			0:
				//初始化
				IF NOT EDTP2S4B_STEP[0].done THEN
					EDTXV0724.control.auto_operate := TRUE;
					EDTAV0702B.control.auto_operate := TRUE;
					EDTAV0702A.control.auto_operate := TRUE;
					EDTXV0716.control.auto_operate := TRUE;
					EDTR12B.control.auto_operate := TRUE;
					EDTTV0703C.control.auto_operate := TRUE;
					EDTTV0703D.control.auto_operate := TRUE;
					EDTTV0703E.control.auto_operate := TRUE;
					EDTTV0703F.control.auto_operate := TRUE;
					EDTFVT0703.control.auto_operate := TRUE;
					EDTXV0719.control.auto_operate := TRUE;
					EDTXV0718.control.auto_operate := TRUE;
					EDTTV0703A.control.auto_operate := TRUE;
					EDTTV0703B.control.auto_operate := TRUE;
					EDTXV0722.control.auto_operate := TRUE;
					EDTXV0723.control.auto_operate := TRUE;
					EDTXV0715.control.auto_operate := TRUE;
					EDTP2S4B_STEP[0].done := TRUE;
				END_IF;
			1:
				//手动分层，完成后点确认
			2:
				//除前馏
				R12B_process1 := TRUE;
				EDTP2S4B_STEP[2].done := TRUE;
			3:
				IF NOT R12B_process1 THEN
					EDTP2S4B_STEP[3].done := TRUE;
				END_IF;
			4:
				//转移确认V19空
			5:
				TON_70.PT := DINT_TO_TIME(EDTP2S4_PARA_T5 * 60 * 1000);
				EDTXV0722.input.auto_open_signal := TRUE;
				IF EDTXV0722.input.open_feedback_state THEN
					TON_70.IN := TRUE;
				END_IF;
				IF TON_70.Q THEN
					TON_70.IN := FALSE;
					EDTP2S4B_STEP[5].done := TRUE;
				END_IF;
				TON_70();
			6:
				//确认R12空
			7:
				TON_71.PT := DINT_TO_TIME(EDTP2S4_PARA_T6 * 60 * 1000);
				EDTXV0722.input.auto_open_signal := FALSE;
				IF EDTXV0722.input.close_feedback_state THEN
					EDTXV0724.input.auto_open_signal := TRUE;
					EDTAV0702A.input.auto_open_signal := TRUE;
				END_IF;
				IF EDTXV0724.input.open_feedback_state AND EDTAV0702A.input.open_feedback_state THEN
					TON_71.IN := TRUE;
				END_IF;
				IF TON_71.Q THEN
					TON_71.IN := FALSE;
					EDTP2S4B_STEP[7].done := TRUE;
				END_IF;
				TON_71();
			8:
				//确认R06空
			9:
				R12B_process := TRUE;
				EDTAV0702A.input.auto_open_signal := FALSE;
				IF EDTAV0702A.input.close_feedback_state THEN
					EDTXV0724.input.auto_open_signal := FALSE;
					IF EDTXV0724.input.close_feedback_state THEN
						EDTXV0723.input.auto_open_signal := TRUE;
						IF EDTXV0723.input.open_feedback_state THEN
							EDTXV0715.input.auto_open_signal := TRUE;
							EDTP2S4B_STEP[9].done := TRUE;
						END_IF;
					END_IF;
				END_IF;
			10:
				//确认转移完毕
			11:
				EDTXV0723.input.auto_open_signal := FALSE;
				EDTXV0715.input.auto_open_signal := FALSE;
				EDTAV0702B.input.auto_open_signal := TRUE;
				EDTXV0724.input.auto_open_signal := TRUE;
				IF EDTXV0723.input.close_feedback_state AND EDTXV0724.input.open_feedback_state AND EDTAV0702B.input.open_feedback_state THEN
					EDTP2S4B_STEP[11].done := TRUE;
				END_IF;
			12:
				//V06-->V22确认转移完毕
			13:
				EDTAV0702B.input.auto_open_signal := FALSE;
				EDTXV0724.input.auto_open_signal := FALSE;
				IF EDTXV0724.input.close_feedback_state AND EDTAV0702B.input.close_feedback_state THEN
					EDTP2S4B_STEP[13].done := TRUE;
				END_IF;
			14:
				IF NOT R12B_process THEN
					EDTP2S4B_STEP[14].done := TRUE;
				END_IF;
			15:
			//转移
		END_CASE;
	END_IF;

	//除前馏
	IF R12B_process1 THEN
		CASE R12B_process1_step OF
			0:
				MTBasicsPID_9.Enable := FALSE;
				EDTXV0716.input.auto_open_signal := TRUE;
				EDTR12B.input.auto_run_signal := TRUE;
				EDTXV0719.input.auto_open_signal := FALSE;
				EDTXV0718.input.auto_open_signal := FALSE;
				EDTFVT0703.input.auto_degree_set := 0.0;
				IF EDTXV0716.input.open_feedback_state AND EDTR12B.input.run_feedback AND EDTXV0719.input.close_feedback_state AND EDTXV0718.input.close_feedback_state THEN
					R12B_process1_step := 1;
				END_IF;
			1:
				HeatPot_6(ST1 := DINT_TO_TIME(EDTP2S4_PARA_T2 * 1000),
				ST2 := DINT_TO_TIME(EDTP2S4_PARA_T3 * 1000),
				V3 := EDTTV0703C,
				V4 := EDTTV0703D,
				V5 := EDTTV0703E,
				V6 := EDTTV0703F,
				done := R12B_process1_step_1_done);
				IF R12B_process1_step_1_done THEN
					R12B_process1_step_1_done := FALSE;
					R12B_process1_step := 2;
				END_IF;
			2:
				IF EDTTIT0703.status.value >= EDTP2S4_PARA_Temp1 THEN
					EDTTV0703C.input.auto_open_signal := FALSE;
					IF EDTTV0703C.input.close_feedback_state THEN
						R12B_process1_step := 3;
					END_IF;
				END_IF;
			3:
				TON_72.PT := DINT_TO_TIME(EDTP2S4_PARA_T4 * 60 * 1000);
				IF EDTTIT0704.status.value >= EDTP2S4_PARA_Temp4 THEN
					TON_72.IN := TRUE;
				END_IF;
				IF TON_72.Q THEN
					TON_72.IN := FALSE;
					R12B_process1_step := 4;
				END_IF;
			4:
				MTBasicsPID_9.Enable := TRUE;
				EDTXV0718.input.auto_open_signal := FALSE;
				IF EDTXV0718.input.close_feedback_state THEN
					EDTXV0719.input.auto_open_signal := TRUE;
					IF EDTXV0719.input.open_feedback_state THEN
						//EDTFVT0703.input.auto_degree_set := EDTP2S4B_PARA_O1;
						R12B_process1_step := 5;
					END_IF;
				END_IF;
			5:
				TON_72.PT := DINT_TO_TIME(EDTP2S4_PARA_T7 * 1000);
				IF EDTTIT0704.status.value >= EDTP2S4_PARA_Temp2 THEN
					EDTTV0703D.input.auto_open_signal := FALSE;
					IF EDTTV0703D.input.close_feedback_state THEN
						EDTTV0703E.input.auto_open_signal := FALSE;
						EDTTV0703F.input.auto_open_signal := TRUE;
						//IF EDTTV0703E.input.close_feedback_state AND EDTTV0703F.input.open_feedback_state THEN
							TON_72.IN := TRUE;
						//END_IF;
					END_IF;
				END_IF;
				IF TON_72.Q THEN
					TON_72.IN := FALSE;
					R12B_process1_step := 6;
				END_IF;
			6:
				EDTTV0703F.input.auto_open_signal := FALSE;
				IF EDTTV0703F.input.close_feedback_state THEN
					EDTTV0703A.input.auto_open_signal := TRUE;
					IF EDTTV0703A.input.open_feedback_state THEN
						EDTTV0703B.input.auto_open_signal := TRUE;
						R12B_process1_step := 7;
					END_IF;
				END_IF;
			7:
				IF EDTTIT0703.status.value <= EDTP2S4_PARA_Temp3 THEN
					MTBasicsPID_9.Enable := FALSE;
					EDTTV0703B.input.auto_open_signal := FALSE;
					EDTTV0703A.input.auto_open_signal := FALSE;
					EDTR12B.input.auto_run_signal := FALSE;
					EDTXV0716.input.auto_open_signal := FALSE;
					EDTFVT0703.input.auto_degree_set := 100.0;
				END_IF;
				IF EDTTV0703A.input.close_feedback_state AND EDTTV0703B.input.close_feedback_state AND (NOT EDTR12B.input.run_feedback) AND EDTXV0716.input.close_feedback_state THEN
					R12B_process1 := FALSE;
					R12B_process1_step := 0;
				END_IF;
		END_CASE;
		TON_72();
	END_IF;

	//甲醇水蒸馏
	IF R12B_process THEN
		CASE R12B_process_step OF
			0:
				//甲醇水蒸馏准备
				MTBasicsPID_9.Enable := FALSE;
				EDTXV0719.input.auto_open_signal := FALSE;
				EDTXV0718.input.auto_open_signal := FALSE;
				EDTXV0716.input.auto_open_signal := TRUE;
				EDTR12B.input.auto_run_signal := TRUE;
				EDTFVT0703.input.auto_degree_set := 0.0;
				IF EDTXV0716.input.open_feedback_state AND EDTR12B.input.run_feedback AND EDTXV0719.input.close_feedback_state AND EDTXV0718.input.close_feedback_state THEN
					R12B_process_step := 1;
				END_IF;
			1:
				HeatPot_10(ST1 := DINT_TO_TIME(EDTP2S4_PARA_T2 * 1000),
				ST2 := DINT_TO_TIME(EDTP2S4_PARA_T3 * 1000),
				V3 := EDTTV0703C,
				V4 := EDTTV0703D,
				V5 := EDTTV0703E,
				V6 := EDTTV0703F,
				done := R12B_process_step_1_done);
				IF R12B_process_step_1_done THEN
					R12B_process_step_1_done := FALSE;
					R12B_process_step := 2;
				END_IF;
			2:
				IF EDTTIT0703.status.value >= EDTP2S4_PARA_Temp1 THEN
					EDTTV0703C.input.auto_open_signal := FALSE;
					IF EDTTV0703C.input.close_feedback_state THEN
						R12B_process_step := 3;
					END_IF;
				END_IF;
			3:
				TON_75.PT := DINT_TO_TIME(EDTP2S4_PARA_T4 * 60 * 1000);
				IF EDTTIT0704.status.value >= EDTP2S4_PARA_Temp4 THEN
					TON_75.IN := TRUE;
				END_IF;
				IF TON_75.Q THEN
					TON_75.IN := FALSE;
					R12B_process_step := 4;
				END_IF;
			4:
				MTBasicsPID_9.Enable := TRUE;
				EDTXV0718.input.auto_open_signal := FALSE;
				IF EDTXV0718.input.close_feedback_state THEN
					EDTXV0719.input.auto_open_signal := TRUE;
					IF EDTXV0719.input.open_feedback_state THEN
						//EDTFVT0703.input.auto_degree_set := EDTP2S4B_PARA_O2;
						R12B_process_step := 5;
					END_IF;
				END_IF;
			5:
				IF EDTTIT0704.status.value >= EDTP2S4_PARA_Temp5 THEN
					EDTXV0719.input.auto_open_signal := FALSE;
					IF EDTXV0719.input.close_feedback_state THEN
						EDTXV0718.input.auto_open_signal := TRUE;
						IF EDTXV0718.input.open_feedback_state THEN
							//EDTFVT0703.input.auto_degree_set := EDTP2S4B_PARA_O3;
							R12B_process_step := 6;
						END_IF;
					END_IF;
				END_IF;
			6:
				TON_75.PT := DINT_TO_TIME(EDTP2S4_PARA_T7 * 1000);
				IF EDTTIT0704.status.value >= EDTP2S4_PARA_Temp6 THEN
					EDTTV0703D.input.auto_open_signal := FALSE;
					IF EDTTV0703D.input.close_feedback_state THEN
						EDTTV0703E.input.auto_open_signal := FALSE;
						EDTTV0703F.input.auto_open_signal := TRUE;
						//IF EDTTV0703E.input.close_feedback_state AND EDTTV0703F.input.open_feedback_state THEN
							TON_75.IN := TRUE;
						//END_IF;
					END_IF;
				END_IF;
				IF TON_75.Q THEN
					TON_75.IN := FALSE;
					R12B_process_step := 7;
				END_IF;
			7:
				EDTTV0703F.input.auto_open_signal := FALSE;
				IF EDTTV0703F.input.close_feedback_state THEN
					EDTTV0703A.input.auto_open_signal := TRUE;
					IF EDTTV0703A.input.open_feedback_state THEN
						EDTTV0703B.input.auto_open_signal := TRUE;
						R12B_process_step := 8;
					END_IF;
				END_IF;
			8:
				IF EDTTIT0703.status.value <= EDTP2S4_PARA_Temp7 THEN
					MTBasicsPID_9.Enable := FALSE;
					EDTTV0703B.input.auto_open_signal := FALSE;
					EDTTV0703A.input.auto_open_signal := FALSE;
					EDTR12B.input.auto_run_signal := FALSE;
					EDTXV0716.input.auto_open_signal := FALSE;
					EDTFVT0703.input.auto_degree_set := 100.0;
				END_IF;
				IF EDTTV0703A.input.close_feedback_state AND EDTTV0703B.input.close_feedback_state AND (NOT EDTR12B.input.run_feedback) AND EDTXV0716.input.close_feedback_state THEN
					R12B_process := FALSE;
					R12B_process_step := 0;
				END_IF;
		END_CASE;
		TON_75();
	END_IF;

	R_TRIG_1(CLK := EDTFVT0703.status.auto_mode);
	IF R_TRIG_1.Q THEN
		MTBasicsPID_9.Enable := TRUE;
	END_IF;
	F_TRIG_1(CLK := EDTFVT0703.status.auto_mode);
	IF F_TRIG_1.Q THEN
		MTBasicsPID_9.Enable := FALSE;
	END_IF;
	//FVT0703 pid调节
	//	MTBasicsPID_9.Enable := TRUE;
	MTBasicsPID_9.PIDParameters.Gain := EDTPid0703Para.gain;
	MTBasicsPID_9.PIDParameters.IntegrationTime := EDTPid0703Para.integration_time;
	MTBasicsPID_9.PIDParameters.DerivativeTime := EDTPid0703Para.derivative_time;
	MTBasicsPID_9.MinOut := 0.0;
	MTBasicsPID_9.MaxOut := 100.0;
	MTBasicsPID_9.SetValue := EDTPid0703Para.set_value;
	MTBasicsPID_9.ActValue := EDTFIT0703.flowrate;
	MTBasicsPID_9.Update := EDTPid0703.update;
	MTBasicsPID_9();
	EDTPid0703.out := MTBasicsPID_9.Out;
	IF MTBasicsPID_9.Active THEN
		EDTFVT0703.input.auto_degree_set := MTBasicsPID_9.Out + EDTPid0703Para.min_out;
		//	ELSE
		//		EDTFVT0703.input.auto_degree_set := 0.0;
	END_IF;
	IF MTBasicsPID_9.UpdateDone THEN
		EDTPid0703.update := FALSE;
	END_IF;

	//人工确认步骤可用
	IF (EDTP2S4B.status.run_state) AND (NOT EDTP2S4B_STEP[EDTP2S4B.status.run_step].done AND ((EDTP2S4B.status.run_step = 1) OR (EDTP2S4B.status.run_step = 4)
		OR (EDTP2S4B.status.run_step = 6) OR (EDTP2S4B.status.run_step = 8) OR (EDTP2S4B.status.run_step = 10) OR (EDTP2S4B.status.run_step = 12) OR (EDTP2S4B.status.run_step = 15))) THEN
		EDTP2S4B.status.confirm_enable := TRUE;
	ELSE
		EDTP2S4B.status.confirm_enable := FALSE;
	END_IF;

END_ACTION

(* ---- EDTP3S1A_ACTION.st ---- *)
ACTION P3S1A_ACT:
	//设定时间
	FOR i := 0 TO EDTP3S1_STEP_NUM DO
		IF EDTP3S1A_ST[i] < T#5s THEN
			EDTP3S1A_ST[i] := T#5s;
		END_IF;
		EDTP3S1A_STEP[i].set_time := EDTP3S1A_ST[i];
	END_FOR;

	//流程步骤
	ProcessHandleFC(EDTP3S1A,EDTP3S1A_STEP[0],EDTP3S1_STEP_NUM);

	//object 手自动切换
	IF (EDTP3S1A.status.mode <> 0) AND (NOT EDTP3S1A.auto_mode_edge) THEN
		EDTP3S1A.auto_mode_edge := TRUE;
		EDTP3S1A.manual_mode_edge := FALSE;

		EDTR18A.control.auto_operate := TRUE;
		EDTTV0801C.control.auto_operate := TRUE;
		EDTTV0801E.control.auto_operate := TRUE;
		EDTTV0801D.control.auto_operate := TRUE;
		EDTTV0801B.control.auto_operate := TRUE;
		EDTTV0801A.control.auto_operate := TRUE;
		EDTXV0812.control.auto_operate := TRUE;
		EDTTVT0801.control.auto_operate := TRUE;
		EDTXV0817.control.auto_operate := TRUE;
		EDTXV2107.control.auto_operate := TRUE;
		EDTXV2113.control.auto_operate := TRUE;
		EDTXV2109.control.auto_operate := TRUE;
	END_IF;

	IF (EDTP3S1A.status.mode = 0) AND (NOT EDTP3S1A.manual_mode_edge) THEN
		EDTP3S1A.manual_mode_edge := TRUE;
		EDTP3S1A.auto_mode_edge := FALSE;

		EDTR18A.control.manual_operate := TRUE;
		EDTTV0801C.control.manual_operate := TRUE;
		EDTTV0801E.control.manual_operate := TRUE;
		EDTTV0801D.control.manual_operate := TRUE;
		EDTTV0801B.control.manual_operate := TRUE;
		EDTTV0801A.control.manual_operate := TRUE;
		EDTXV0812.control.manual_operate := TRUE;
		EDTTVT0801.control.manual_operate := TRUE;
		EDTXV0817.control.manual_operate := TRUE;
		EDTXV2107.control.manual_operate := TRUE;
		EDTXV2113.control.manual_operate := TRUE;
		EDTXV2109.control.manual_operate := TRUE;
	END_IF;

	//错误信号停机
	EDTP3S1A.input.error_signal := (EDTR18A.status.motor_status >= 2) OR (EDTTV0801C.status.valve_status >= 2) OR (EDTTV0801E.status.valve_status >= 2) OR
	(EDTTV0801D.status.valve_status >= 2) OR(EDTTV0801B.status.valve_status >= 2) OR (EDTTV0801A.status.valve_status >= 2) OR (EDTXV0812.status.valve_status >= 2);

	IF EDTP3S1A.status.run_state = 1 THEN
		CASE EDTP3S1A.status.run_step OF
			0:
				IF NOT EDTP3S1A_STEP[0].done THEN
					EDTR18A.control.auto_operate := TRUE;
					EDTTV0801C.control.auto_operate := TRUE;
					EDTTV0801E.control.auto_operate := TRUE;
					EDTTV0801D.control.auto_operate := TRUE;
					EDTTV0801B.control.auto_operate := TRUE;
					EDTTV0801A.control.auto_operate := TRUE;
					EDTXV0812.control.auto_operate := TRUE;
					EDTTVT0801.control.auto_operate := TRUE;
					EDTXV0817.control.auto_operate := TRUE;
					EDTXV2107.control.auto_operate := TRUE;
					EDTXV2113.control.auto_operate := TRUE;
					EDTXV2109.control.auto_operate := TRUE;
					IF EDTXV0801.input.close_feedback_state AND EDTXV0806.input.close_feedback_state AND EDTXV0804.input.close_feedback_state AND EDTFQV0801.input.close_feedback_state
						AND EDTXV0814.input.close_feedback_state AND EDTXV0822.input.close_feedback_state AND EDTXV0817.input.close_feedback_state THEN
						EDTP3S1A_STEP[0].done := TRUE;
					END_IF;
				END_IF;
			1:
				//醚化
				CASE p3_step1_1a OF
					0:
						IF NOT EDTP3S1A_STEP[1].done THEN
							p3_step1_1a := 1;
						END_IF;
					1:
						TON_0.IN := FALSE;
						TON_46.IN := FALSE;
						temp_decrease := FALSE;
						FOR i := 0 TO 50 DO
							EDTTIT0801_avg_record[i] := 0;
						END_FOR;
						EDTTIT0801_avg := 0;
						n := 0;
						temp_offset := 0;
						offset := 0;
						EDTPIT0803_record[0] := REAL_TO_INT(EDTPIT0803_PARA.upper_range * 100);
						EDTPIT0803_record[1] := REAL_TO_INT(EDTPIT0803_PARA.upper_range * 100);
						EDTPIT0803_record[2] := REAL_TO_INT(EDTPIT0803_PARA.upper_range * 100);
						EDTTIT0801_record[0] := REAL_TO_INT(EDTTIT0801_PARA.upper_range * 100);
						EDTTIT0801_record[1] := REAL_TO_INT(EDTTIT0801_PARA.upper_range * 100);
						EDTTIT0801_record[2] := REAL_TO_INT(EDTTIT0801_PARA.upper_range * 100);
						EDTR18A.input.auto_run_signal := TRUE;
						IF EDTR18A.input.run_feedback THEN
							p3_step1_1a := 2;
						END_IF;
					2:
						TON_0.PT := DINT_TO_TIME(EDTP3S1_PARA_T2 * 1000);
						EDTTV0801E.input.auto_open_signal := TRUE;
						IF EDTTV0801E.input.open_feedback_state THEN
							EDTXV0812.input.auto_open_signal := TRUE;
							TON_0.IN := TRUE;
						END_IF;
						IF TON_0.Q THEN
							TON_0.IN := FALSE;
							p3_step1_1a := 3;
						END_IF;
					3:
						//每两秒采集一个数据，连续采集3个，连续下降则判定值开始下降
						TON_0.PT := DINT_TO_TIME(EDTP3S1_PARA_T1 * 1000);
						TON_0.IN := TRUE;
						IF TON_0.Q THEN
							TON_0.IN := FALSE;
							EDTPIT0803_record[offset] := REAL_TO_INT(EDTPIT0803.status.value * 100);
							offset := offset + 1;
						END_IF;
						IF offset > 2 THEN
							offset := 0;
						END_IF;
						IF (EDTPIT0803_record[0] > EDTPIT0803_record[1]) AND (EDTPIT0803_record[1] > EDTPIT0803_record[2]) THEN
							p3_step1_1a := 4;
						END_IF;
					4:
						IF EDTPIT0803.status.value <= EDTP3S1_PARA_P3 THEN
							EDTXV0812.input.auto_open_signal := FALSE;
						END_IF;
						IF EDTPIT0803.status.value <= EDTP3S1_PARA_P4 THEN
							EDTTV0801E.input.auto_open_signal := FALSE;
							EDTTV0801D.input.auto_open_signal := TRUE;
							IF EDTTV0801D.input.open_feedback_state THEN
								EDTTV0801C.input.auto_open_signal := TRUE;
								EDTPid0801Para.set_value := EDTP3S1_PARA_Temp1;
								MTBasicsPID_0.Enable := TRUE;
								p3_step1_1a := 5;
							END_IF;
						END_IF;
					5:
						//大于125℃计时5h
						TON_0.PT := DINT_TO_TIME(EDTP3S1_PARA_T3 * 60 * 1000);
						IF EDTTIT0801.status.value >= EDTP3S1_PARA_Temp2 THEN
							TON_0.IN := TRUE;
						END_IF;
						IF EDTTIT0801.status.value >= EDTP3S1_PARA_Temp1 THEN
							EDTTV0801C.input.auto_open_signal := FALSE;
							R18A_start := TRUE;
							p3_step1_1a := 6;
						END_IF;
					6:
						TON_0.PT := DINT_TO_TIME(EDTP3S1_PARA_T3 * 60 * 1000);
						IF TON_0.Q THEN
							TON_0.IN := FALSE;
							p3_step1_1a := 7;
						END_IF;
					7:
						//复位温控
						R18A_start := FALSE;
						temp_h_flag := FALSE;
						R18A_step_1 := 0;
						press_h_flag := FALSE;
						R18A_step_2 := 0;
						temp_l_flag := FALSE;
						R18A_step_3 := 0;

						EDTTV0801C.input.auto_open_signal := FALSE;
						EDTTV0801E.input.auto_open_signal := FALSE;
						EDTTV0801D.input.auto_open_signal := FALSE;
						EDTXV0812.input.auto_open_signal := FALSE;
						IF EDTTV0801C.input.close_feedback_state AND EDTTV0801E.input.close_feedback_state AND EDTTV0801D.input.close_feedback_state THEN
							p3_step1_1a := 8;
						END_IF;
					8:
						MTBasicsPID_0.Enable := FALSE;
						EDTTV0801A.input.auto_open_signal := TRUE;
						EDTTV0801B.input.auto_open_signal := TRUE;
						IF EDTTV0801A.input.open_feedback_state AND EDTTV0801B.input.open_feedback_state THEN
							p3_step1_1a := 9;
						END_IF;
					9:
						IF EDTTIT0801.status.value <= EDTP3S1_PARA_Temp3 THEN
							EDTTV0801B.input.auto_open_signal := FALSE;
							EDTTV0801A.input.auto_open_signal := FALSE;
							EDTP3S1A_STEP[1].done := TRUE;
							p3_step1_1a := 0;
						END_IF;
				END_CASE;
				TON_0();
			2:
				IF NOT EDTP3S2C.status.run_state THEN
					EDTXV2109.input.auto_open_signal := FALSE;
					IF EDTXV2109.input.close_feedback_state THEN
						EDTXV0817.input.auto_open_signal := TRUE;
						EDTXV2107.input.auto_open_signal := TRUE;
						EDTXV2113.input.auto_open_signal := TRUE;
						IF EDTPIT0801.status.value <= EDTP3S1_PARA_P5 THEN
							EDTP3S1A_STEP[2].done := TRUE;
						END_IF;
					END_IF;
				END_IF;
			3:
				//人工转移
		END_CASE;
	END_IF;

	//R18A控温、控压
	//=======================================================================================================
	IF R18A_start THEN
		//每两秒采集一个数据，连续采集3个，连续下降则判定为温度开始下降
		IF EDTP3S1_PARA_T1 >= 4 THEN
			EDTP3S1_PARA_T1 := 4;
		END_IF;
		IF EDTP3S1_PARA_T1 <= 1 THEN
			EDTP3S1_PARA_T1 := 1;
		END_IF;
		TON_46.PT := DINT_TO_TIME(EDTP3S1_PARA_T1 * 1000);
		TON_46.IN := TRUE;
		EDTTIT0801_avg_record[n] := EDTTIT0801.status.value;
		n := n + 1;
		IF TON_46.Q THEN
			TON_46.IN := FALSE;
			FOR i := 0 TO n DO
				EDTTIT0801_avg := EDTTIT0801_avg_record[i] + EDTTIT0801_avg;
			END_FOR;
			EDTTIT0801_record[temp_offset] := REAL_TO_INT(EDTTIT0801_avg * 100 / n);
			FOR i := 0 TO 50 DO
				EDTTIT0801_avg_record[i] := 0;
			END_FOR;
			EDTTIT0801_avg := 0;
			n := 0;
			//	EDTTIT0801_record[temp_offset] := REAL_TO_INT(EDTTIT0801.status.value * 100);
			temp_offset := temp_offset + 1;
		END_IF;
		IF temp_offset > 3 THEN
			temp_offset := 0;
		END_IF;
		IF (EDTTIT0801_record[0] > EDTTIT0801_record[1]) AND (EDTTIT0801_record[1] > EDTTIT0801_record[2]) AND
			(EDTTIT0801_record[0] <> REAL_TO_INT(EDTTIT0801_PARA.upper_range * 100)) AND
			(EDTTIT0801_record[1] <> REAL_TO_INT(EDTTIT0801_PARA.upper_range * 100)) AND
			(EDTTIT0801_record[2] <> REAL_TO_INT(EDTTIT0801_PARA.upper_range * 100)) THEN
			temp_decrease := TRUE;
		ELSE
			temp_decrease := FALSE;
		END_IF;
		TON_46();

		IF EDTTIT0801.status.value >= EDTP3S1_PARA_Temp4 AND (NOT temp_h_flag) AND (R18A_step_2 = 0) AND (R18A_step_3 = 0) THEN
			R18A_step_1 := 1;
			temp_h_flag := TRUE;
		END_IF;
		IF EDTPIT0801.status.value >= EDTP3S1_PARA_P1 AND (NOT press_h_flag) AND (R18A_step_1 = 0) AND (R18A_step_3 = 0) THEN
			R18A_step_2 := 1;
			press_h_flag := TRUE;
		END_IF;
		IF (EDTTIT0801.status.value <= EDTP3S1_PARA_Temp5) AND (NOT temp_l_flag) AND (R18A_step_1 = 0) AND (R18A_step_2 = 0) THEN
			R18A_step_3 := 1;
			temp_l_flag := TRUE;
		END_IF;
	END_IF;

	//温度上限
	CASE R18A_step_1 OF
		0:
			//idle
		1:
			TON_25.IN := FALSE;
			EDTPIT0803_record[0] := REAL_TO_INT(EDTPIT0803_PARA.upper_range * 100);
			EDTPIT0803_record[1] := REAL_TO_INT(EDTPIT0803_PARA.upper_range * 100);
			EDTPIT0803_record[2] := REAL_TO_INT(EDTPIT0803_PARA.upper_range * 100);
			EDTTIT0801_record[0] := REAL_TO_INT(EDTTIT0801_PARA.upper_range * 100);
			EDTTIT0801_record[1] := REAL_TO_INT(EDTTIT0801_PARA.upper_range * 100);
			EDTTIT0801_record[2] := REAL_TO_INT(EDTTIT0801_PARA.upper_range * 100);
			R18A_step_1 := 2;
		2:
			EDTTV0801E.input.auto_open_signal := TRUE;
			TON_25.PT := DINT_TO_TIME(EDTP3S1_PARA_T4 * 1000);
			TON_25.IN := TRUE;
			IF TON_25.Q THEN
				TON_25.IN := FALSE;
				R18A_step_1 := 3;
			END_IF;
		3:
			EDTTV0801E.input.auto_open_signal := FALSE;
			EDTTV0801D.input.auto_open_signal := FALSE;
			R18A_step_1 := 4;
		4:
			EDTTV0801A.input.auto_open_signal := TRUE;
			IF EDTTV0801A.input.open_feedback_state THEN
				EDTTV0801B.input.auto_open_signal := TRUE;
			END_IF;
			IF EDTTV0801B.input.open_feedback_state AND EDTTV0801A.input.open_feedback_state THEN
				R18A_step_1 := 5;
			END_IF;
		5:
			//每两秒采集一个数据，连续采集3个，连续下降则判定为温度开始下降
			IF temp_decrease THEN
				R18A_step_1 := 6;
			END_IF;
		6:
			EDTTV0801B.input.auto_open_signal := FALSE;
			IF EDTTV0801B.input.close_feedback_state THEN
				EDTTV0801A.input.auto_open_signal := FALSE;
			END_IF;
			IF EDTTV0801A.input.close_feedback_state AND EDTTV0801B.input.close_feedback_state THEN
				R18A_step_1 := 7;
			END_IF;
		7:
			EDTTV0801E.input.auto_open_signal := TRUE;
			IF EDTTV0801E.input.open_feedback_state THEN
				EDTXV0812.input.auto_open_signal := TRUE;
				R18A_step_1 := 8;
			END_IF;
		8:
			TON_25.PT := DINT_TO_TIME(EDTP3S1_PARA_T2 * 1000);
			TON_25.IN := TRUE;
			IF TON_25.Q THEN
				TON_25.IN := FALSE;
				R18A_step_1 := 9;
			END_IF;
		9:
			//每两秒采集一个数据，连续采集3个，连续下降则判定值开始下降
			TON_25.PT := DINT_TO_TIME(EDTP3S1_PARA_T1 * 1000);
			TON_25.IN := TRUE;
			IF TON_25.Q THEN
				TON_25.IN := FALSE;
				EDTPIT0803_record[offset] := REAL_TO_INT(EDTPIT0803.status.value * 100);
				offset := offset + 1;
			END_IF;
			IF offset > 2 THEN
				offset := 0;
			END_IF;
			IF (EDTPIT0803_record[0] > EDTPIT0803_record[1]) AND (EDTPIT0803_record[1] > EDTPIT0803_record[2]) THEN
				R18A_step_1 := 10;
			END_IF;
		10:
			IF EDTPIT0803.status.value <= EDTP3S1_PARA_P3 THEN
				EDTXV0812.input.auto_open_signal := FALSE;
				temp_h_flag := FALSE;
				R18A_step_1 := 0;
			END_IF;
	END_CASE;
	TON_25();

	//压力上限
	CASE R18A_step_2 OF
		0:
			//idle
		1:
			EDTPIT0803_record[0] := REAL_TO_INT(EDTPIT0803_PARA.upper_range * 100);
			EDTPIT0803_record[1] := REAL_TO_INT(EDTPIT0803_PARA.upper_range * 100);
			EDTPIT0803_record[2] := REAL_TO_INT(EDTPIT0803_PARA.upper_range * 100);
			TON_27.IN := FALSE;
			EDTTV0801E.input.auto_open_signal := FALSE;
			EDTTV0801D.input.auto_open_signal := FALSE;
			IF EDTTV0801E.input.close_feedback_state AND EDTTV0801D.input.close_feedback_state AND EDTTV0801C.input.close_feedback_state THEN
				R18A_step_2 := 2;
			END_IF;
		2:
			EDTTV0801A.input.auto_open_signal := TRUE;
			IF EDTTV0801A.input.open_feedback_state THEN
				EDTTV0801B.input.auto_open_signal := TRUE;
			END_IF;
			IF EDTTV0801B.input.open_feedback_state AND EDTTV0801A.input.open_feedback_state THEN
				R18A_step_2 := 3;
			END_IF;
		3:
			IF EDTPIT0801.status.value <= EDTP3S1_PARA_P2 THEN
				R18A_step_2 := 4;
			END_IF;
		4:
			EDTTV0801B.input.auto_open_signal := FALSE;
			IF EDTTV0801B.input.close_feedback_state THEN
				EDTTV0801A.input.auto_open_signal := FALSE;
			END_IF;
			IF EDTTV0801A.input.close_feedback_state AND EDTTV0801B.input.close_feedback_state THEN
				R18A_step_2 := 5;
			END_IF;
		5:
			EDTTV0801E.input.auto_open_signal := TRUE;
			IF EDTTV0801E.input.open_feedback_state THEN
				EDTXV0812.input.auto_open_signal := TRUE;
				R18A_step_2 := 6;
			END_IF;
		6:
			TON_27.PT := DINT_TO_TIME(EDTP3S1_PARA_T2 * 1000);
			TON_27.IN := TRUE;
			IF TON_27.Q THEN
				TON_27.IN := FALSE;
				R18A_step_2 := 7;
			END_IF;
		7:
			//每两秒采集一个数据，连续采集3个，连续下降则判定值开始下降
			TON_27.PT := DINT_TO_TIME(EDTP3S1_PARA_T1 * 1000);
			TON_27.IN := TRUE;
			IF TON_27.Q THEN
				TON_27.IN := FALSE;
				EDTPIT0803_record[offset] := REAL_TO_INT(EDTPIT0803.status.value * 100);
				offset := offset + 1;
			END_IF;
			IF offset > 2 THEN
				offset := 0;
			END_IF;
			IF (EDTPIT0803_record[0] > EDTPIT0803_record[1]) AND (EDTPIT0803_record[1] > EDTPIT0803_record[2]) THEN
				R18A_step_2 := 8;
			END_IF;
		8:
			IF EDTPIT0803.status.value <= EDTP3S1_PARA_P3 THEN
				EDTXV0812.input.auto_open_signal := FALSE;
				press_h_flag := FALSE;
				R18A_step_2 := 0;
			END_IF;
	END_CASE;
	TON_27();

	//温度低限
	CASE R18A_step_3 OF
		0:
			//idle
		1:
			EDTTV0801E.input.auto_open_signal := FALSE;
			EDTXV0812.input.auto_open_signal := FALSE;
			EDTTV0801C.input.auto_open_signal := TRUE;
			EDTTV0801D.input.auto_open_signal := TRUE;
			R18A_step_3 := 2;
		2:
			IF EDTTIT0801.status.value >= EDTP3S1_PARA_Temp1 THEN
				R18A_step_3 := 3;
			END_IF;
		3:
			EDTTV0801C.input.auto_open_signal := FALSE;
			EDTTV0801D.input.auto_open_signal := FALSE;
			EDTTV0801E.input.auto_open_signal := TRUE;
			R18A_step_3 := 4;
		4:
			temp_l_flag := FALSE;
			R18A_step_3 := 0;
	END_CASE;

	IF r20_transfer THEN
		CASE r20_transfer_step OF
			0:
				EDTXV2109.control.auto_operate := TRUE;
				EDTXV2107.control.auto_operate := TRUE;
				EDTXV2111.control.auto_operate := TRUE;
				r20_transfer_step := 1;
			1:
				EDTXV2109.input.auto_open_signal := TRUE;
				EDTXV2107.input.auto_open_signal := TRUE;
				EDTXV2111.input.auto_open_signal := TRUE;
				r20_transfer_step := 2;
			2:
				r20_transfer_step := 0;
				r20_transfer := FALSE;
		END_CASE;
	END_IF;
	IF r17_transfer THEN
		CASE r17_transfer_step OF
			0:
				EDTXV0925.control.auto_operate := TRUE;
				EDTXV0902.control.auto_operate := TRUE;
				EDTXV0912.control.auto_operate := TRUE;
				EDTTV0902B.control.auto_operate := TRUE;
				EDTTV0904B.control.auto_operate := TRUE;
				r17_transfer_step := 1;
			1:
				EDTXV0925.input.auto_open_signal := TRUE;
				EDTXV0902.input.auto_open_signal := TRUE;
				EDTXV0912.input.auto_open_signal := TRUE;
				EDTTV0902B.input.auto_open_signal := TRUE;
				EDTTV0904B.input.auto_open_signal := TRUE;
				r17_transfer_step := 2;
			2:
				r17_transfer_step := 0;
				r17_transfer := FALSE;
		END_CASE;
	END_IF;
	//=======================================================================================================
	//pid 温度调节

	R_TRIG_2(CLK := EDTTVT0801.status.auto_mode);
	IF R_TRIG_2.Q THEN
		MTBasicsPID_0.Enable := TRUE;
	END_IF;
	F_TRIG_2(CLK := EDTTVT0801.status.auto_mode);
	IF F_TRIG_2.Q THEN
		MTBasicsPID_0.Enable := FALSE;
	END_IF;

	//MTBasicsPID_0.Enable := TRUE;
	//MTBasicsPID_0.Invert := TRUE;
	MTBasicsPID_0.PIDParameters.Gain := EDTPid0801Para.gain;
	MTBasicsPID_0.PIDParameters.IntegrationTime := EDTPid0801Para.integration_time;
	MTBasicsPID_0.PIDParameters.DerivativeTime := EDTPid0801Para.derivative_time;
	MTBasicsPID_0.MinOut := 0.0;
	MTBasicsPID_0.MaxOut := 100.0;
	MTBasicsPID_0.SetValue := EDTPid0801Para.set_value;
	MTBasicsPID_0.ActValue := EDTTIT0801.status.value;
	MTBasicsPID_0.Update := EDTPid0801.update;
	MTBasicsPID_0();
	EDTPid0801.out := MTBasicsPID_0.Out;
	IF MTBasicsPID_0.Active THEN
		EDTTVT0801.input.auto_degree_set := MTBasicsPID_0.Out;
	ELSE
		EDTTVT0801.input.auto_degree_set := 0.0;
	END_IF;
	IF MTBasicsPID_0.UpdateDone THEN
		EDTPid0801.update := FALSE;
	END_IF;

	//人工确认步骤可用
	IF (EDTP3S1A.status.run_state) AND (NOT EDTP3S1A_STEP[EDTP3S1A.status.run_step].done AND ((EDTP3S1A.status.run_step = 3))) THEN
		EDTP3S1A.status.confirm_enable := TRUE;
	ELSE
		EDTP3S1A.status.confirm_enable := FALSE;
	END_IF;
END_ACTION

(* ---- EDTP3S1B_ACTION.st ---- *)
ACTION P3S1B_ACT:
	//设定时间
	FOR i := 0 TO EDTP3S1_STEP_NUM DO
		IF EDTP3S1B_ST[i] < T#5s THEN
			EDTP3S1B_ST[i] := T#5s;
		END_IF;
		EDTP3S1B_STEP[i].set_time := EDTP3S1B_ST[i];
	END_FOR;

	//流程步骤
	ProcessHandleFC(EDTP3S1B,EDTP3S1B_STEP[0],EDTP3S1_STEP_NUM);

	//object 手自动切换
	IF (EDTP3S1B.status.mode <> 0) AND (NOT EDTP3S1B.auto_mode_edge) THEN
		EDTP3S1B.auto_mode_edge := TRUE;
		EDTP3S1B.manual_mode_edge := FALSE;

		EDTR18B.control.auto_operate := TRUE;
		EDTTV0802C.control.auto_operate := TRUE;
		EDTTV0802E.control.auto_operate := TRUE;
		EDTTV0802D.control.auto_operate := TRUE;
		EDTTV0802B.control.auto_operate := TRUE;
		EDTTV0802A.control.auto_operate := TRUE;
		EDTXV0813.control.auto_operate := TRUE;
		EDTTVT0802.control.auto_operate := TRUE;
		EDTXV0818.control.auto_operate := TRUE;
		EDTXV0902.control.auto_operate := TRUE;
		EDTXV0912.control.auto_operate := TRUE;
		EDTTV0902A.control.auto_operate := TRUE;
		EDTTV0904A.control.auto_operate := TRUE;
		EDTXV2128.control.auto_operate := TRUE;
		EDTXV0925.control.auto_operate := TRUE;
	END_IF;

	IF (EDTP3S1B.status.mode = 0) AND (NOT EDTP3S1B.manual_mode_edge) THEN
		EDTP3S1B.manual_mode_edge := TRUE;
		EDTP3S1B.auto_mode_edge := FALSE;

		EDTR18B.control.manual_operate := TRUE;
		EDTTV0802C.control.manual_operate := TRUE;
		EDTTV0802E.control.manual_operate := TRUE;
		EDTTV0802D.control.manual_operate := TRUE;
		EDTTV0802B.control.manual_operate := TRUE;
		EDTTV0802A.control.manual_operate := TRUE;
		EDTXV0813.control.manual_operate := TRUE;
		EDTTVT0802.control.manual_operate := TRUE;
		EDTXV0818.control.manual_operate := TRUE;
		EDTXV0902.control.manual_operate := TRUE;
		EDTXV0912.control.manual_operate := TRUE;
		EDTTV0902A.control.manual_operate := TRUE;
		EDTTV0904A.control.manual_operate := TRUE;
		EDTXV2128.control.manual_operate := TRUE;
		EDTXV0925.control.manual_operate := TRUE;
	END_IF;

	//错误信号停机
	EDTP3S1B.input.error_signal := (EDTR18B.status.motor_status >= 2) OR (EDTTV0802C.status.valve_status >= 2) OR (EDTTV0802E.status.valve_status >= 2) OR
	(EDTTV0802D.status.valve_status >= 2) OR(EDTTV0802B.status.valve_status >= 2) OR (EDTTV0802A.status.valve_status >= 2) OR (EDTXV0813.status.valve_status >= 2);

	IF EDTP3S1B.status.run_state = 1 THEN
		CASE EDTP3S1B.status.run_step OF
			0:
				IF NOT EDTP3S1B_STEP[0].done THEN
					EDTR18B.control.auto_operate := TRUE;
					EDTTV0802C.control.auto_operate := TRUE;
					EDTTV0802E.control.auto_operate := TRUE;
					EDTTV0802D.control.auto_operate := TRUE;
					EDTTV0802B.control.auto_operate := TRUE;
					EDTTV0802A.control.auto_operate := TRUE;
					EDTXV0813.control.auto_operate := TRUE;
					EDTTVT0802.control.auto_operate := TRUE;
					EDTXV0818.control.auto_operate := TRUE;
					EDTXV0902.control.auto_operate := TRUE;
					EDTXV0912.control.auto_operate := TRUE;
					EDTTV0902A.control.auto_operate := TRUE;
					EDTTV0904A.control.auto_operate := TRUE;
					EDTXV2128.control.auto_operate := TRUE;
					EDTXV0925.control.auto_operate := TRUE;
					IF EDTXV0807.input.close_feedback_state AND EDTXV0818.input.close_feedback_state AND EDTXV0810.input.close_feedback_state AND EDTFQV0802.input.close_feedback_state
						AND EDTXV0809.input.close_feedback_state AND EDTXV0815.input.close_feedback_state AND EDTXV0823.input.close_feedback_state THEN
						EDTP3S1B_STEP[0].done := TRUE;
					END_IF;
				END_IF;
			1:
				//醚化
				CASE p3_step1_1b OF
					0:
						IF NOT EDTP3S1B_STEP[1].done THEN
							p3_step1_1b := 1;
						END_IF;
					1:
						TON_52.IN := FALSE;
						TON_58.IN := FALSE;
						temp_decrease_0802 := FALSE;
						FOR i := 0 TO 50 DO
							EDTTIT0802_avg_record[i] := 0;
						END_FOR;
						EDTTIT0802_avg := 0;
						m := 0;
						temp_offset_b := 0;
						offset_b := 0;
						EDTPIT0804_record[0] := REAL_TO_INT(EDTPIT0804_PARA.upper_range * 100);
						EDTPIT0804_record[1] := REAL_TO_INT(EDTPIT0804_PARA.upper_range * 100);
						EDTPIT0804_record[2] := REAL_TO_INT(EDTPIT0804_PARA.upper_range * 100);
						EDTTIT0802_record[0] := REAL_TO_INT(EDTTIT0802_PARA.upper_range * 100);
						EDTTIT0802_record[1] := REAL_TO_INT(EDTTIT0802_PARA.upper_range * 100);
						EDTTIT0802_record[2] := REAL_TO_INT(EDTTIT0802_PARA.upper_range * 100);
						EDTR18B.input.auto_run_signal := TRUE;
						IF EDTR18B.input.run_feedback THEN
							p3_step1_1b := 2;
						END_IF;
					2:
						TON_52.PT := DINT_TO_TIME(EDTP3S1_PARA_T2 * 1000);
						EDTTV0802E.input.auto_open_signal := TRUE;
						IF EDTTV0802E.input.open_feedback_state THEN
							EDTXV0813.input.auto_open_signal := TRUE;
							TON_52.IN := TRUE;
						END_IF;
						IF TON_52.Q THEN
							TON_52.IN := FALSE;
							p3_step1_1b := 3;
						END_IF;
					3:
						//每两秒采集一个数据，连续采集3个，连续下降则判定值开始下降
						TON_52.PT := DINT_TO_TIME(EDTP3S1_PARA_T1 * 1000);
						TON_52.IN := TRUE;
						IF TON_52.Q THEN
							TON_52.IN := FALSE;
							EDTPIT0804_record[offset_b] := REAL_TO_INT(EDTPIT0804.status.value * 100);
							offset_b := offset_b + 1;
						END_IF;
						IF offset_b > 2 THEN
							offset_b := 0;
						END_IF;
						IF (EDTPIT0804_record[0] > EDTPIT0804_record[1]) AND (EDTPIT0804_record[1] > EDTPIT0804_record[2]) THEN
							p3_step1_1b := 4;
						END_IF;
					4:
						IF EDTPIT0804.status.value <= EDTP3S1_PARA_P3 THEN
							EDTXV0813.input.auto_open_signal := FALSE;
						END_IF;
						IF EDTPIT0804.status.value <= EDTP3S1_PARA_P4 THEN
							EDTTV0802E.input.auto_open_signal := FALSE;
							EDTTV0802D.input.auto_open_signal := TRUE;
							IF EDTTV0802D.input.open_feedback_state THEN
								EDTTV0802C.input.auto_open_signal := TRUE;
								EDTPid0802Para.set_value := EDTP3S1_PARA_Temp1;
								MTBasicsPID_7.Enable := TRUE;
								p3_step1_1b := 5;
							END_IF;
						END_IF;
					5:
						//大于125℃计时5h
						TON_52.PT := DINT_TO_TIME(EDTP3S1_PARA_T3 * 60 * 1000);
						IF EDTTIT0802.status.value >= EDTP3S1_PARA_Temp2 THEN
							TON_52.IN := TRUE;
						END_IF;
						IF EDTTIT0802.status.value >= EDTP3S1_PARA_Temp1 THEN
							EDTTV0802C.input.auto_open_signal := FALSE;
							R18B_start := TRUE;
							p3_step1_1b := 6;
						END_IF;
					6:
						TON_52.PT := DINT_TO_TIME(EDTP3S1_PARA_T3 * 60 * 1000);
						IF TON_52.Q THEN
							TON_52.IN := FALSE;
							p3_step1_1b := 7;
						END_IF;
					7:
						//复位温控
						R18B_start := FALSE;
						temp_h_flag_b := FALSE;
						R18B_step_1 := 0;
						press_h_flag_b := FALSE;
						R18B_step_2 := 0;
						temp_l_flag_b := FALSE;
						R18B_step_3 := 0;

						EDTTV0802C.input.auto_open_signal := FALSE;
						EDTTV0802E.input.auto_open_signal := FALSE;
						EDTTV0802D.input.auto_open_signal := FALSE;
						EDTXV0813.input.auto_open_signal := FALSE;
						IF EDTTV0802C.input.close_feedback_state AND EDTTV0802E.input.close_feedback_state AND EDTTV0802D.input.close_feedback_state THEN
							p3_step1_1b := 8;
						END_IF;
					8:
						MTBasicsPID_7.Enable := FALSE;
						EDTTV0802A.input.auto_open_signal := TRUE;
						EDTTV0802B.input.auto_open_signal := TRUE;
						IF EDTTV0802A.input.open_feedback_state AND EDTTV0802B.input.open_feedback_state THEN
							p3_step1_1b := 9;
						END_IF;
					9:
						IF EDTTIT0802.status.value <= EDTP3S1_PARA_Temp3 THEN
							EDTTV0802B.input.auto_open_signal := FALSE;
							EDTTV0802A.input.auto_open_signal := FALSE;
							EDTP3S1B_STEP[1].done := TRUE;
							p3_step1_1b := 0;
						END_IF;
				END_CASE;
				TON_52();
			2:
				IF (NOT EDTP3S2A.status.run_state) AND (NOT EDTP3S2B.status.run_state) THEN
					EDTXV0925.input.auto_open_signal := FALSE;
					IF EDTXV0925.input.close_feedback_state THEN
						EDTXV0818.input.auto_open_signal := TRUE;
						EDTXV0902.input.auto_open_signal := TRUE;
						EDTXV0912.input.auto_open_signal := TRUE;
						EDTTV0902A.input.auto_open_signal := TRUE;
						EDTTV0904A.input.auto_open_signal := TRUE;
						EDTXV2128.input.auto_open_signal := TRUE;
						IF EDTPIT0802.status.value <= EDTP3S1_PARA_P5 THEN
							EDTP3S1B_STEP[2].done := TRUE;
						END_IF;
					END_IF;
				END_IF;
			3:
			//人工转移
		END_CASE;
	END_IF;

	//R18B控温、控压
	//=======================================================================================================
	IF R18B_start THEN
		//每两秒采集一个数据，连续采集3个，连续下降则判定为温度开始下降
		IF EDTP3S1_PARA_T1 >= 4 THEN
			EDTP3S1_PARA_T1 := 4;
		END_IF;
		IF EDTP3S1_PARA_T1 <= 1 THEN
			EDTP3S1_PARA_T1 := 1;
		END_IF;
		TON_58.PT := DINT_TO_TIME(EDTP3S1_PARA_T1 * 1000);
		TON_58.IN := TRUE;
		EDTTIT0802_avg_record[m] := EDTTIT0802.status.value;
		m := m + 1;
		IF TON_58.Q THEN
			TON_58.IN := FALSE;
			FOR i := 0 TO m DO
				EDTTIT0802_avg := EDTTIT0802_avg_record[i] + EDTTIT0802_avg;
			END_FOR;
			EDTTIT0802_record[temp_offset_b] := REAL_TO_INT(EDTTIT0802_avg * 100 / m);
			FOR i := 0 TO 50 DO
				EDTTIT0802_avg_record[i] := 0;
			END_FOR;
			EDTTIT0802_avg := 0;
			m := 0;
			//	EDTTIT0802_record[temp_offset_b] := REAL_TO_INT(EDTTIT0802.status.value * 100);
			temp_offset_b := temp_offset_b + 1;
		END_IF;
		IF temp_offset_b > 3 THEN
			temp_offset_b := 0;
		END_IF;
		IF (EDTTIT0802_record[0] > EDTTIT0802_record[1]) AND (EDTTIT0802_record[1] > EDTTIT0802_record[2]) AND
			(EDTTIT0802_record[0] <> REAL_TO_INT(EDTTIT0802_PARA.upper_range * 100)) AND
			(EDTTIT0802_record[1] <> REAL_TO_INT(EDTTIT0802_PARA.upper_range * 100)) AND
			(EDTTIT0802_record[2] <> REAL_TO_INT(EDTTIT0802_PARA.upper_range * 100)) THEN
			temp_decrease_0802 := TRUE;
		ELSE
			temp_decrease_0802 := FALSE;
		END_IF;
		TON_58();

		IF EDTTIT0802.status.value >= EDTP3S1_PARA_Temp4 AND (NOT temp_h_flag_b) AND (R18B_step_2 = 0) AND (R18B_step_3 = 0) THEN
			R18B_step_1 := 1;
			temp_h_flag_b := TRUE;
		END_IF;
		IF EDTPIT0802.status.value >= EDTP3S1_PARA_P1 AND (NOT press_h_flag_b) AND (R18B_step_1 = 0) AND (R18B_step_3 = 0) THEN
			R18B_step_2 := 1;
			press_h_flag_b := TRUE;
		END_IF;
		IF (EDTTIT0802.status.value <= EDTP3S1_PARA_Temp5) AND (NOT temp_l_flag_b) AND (R18B_step_1 = 0) AND (R18B_step_2 = 0) THEN
			R18B_step_3 := 1;
			temp_l_flag_b := TRUE;
		END_IF;
	END_IF;

	//温度上限
	CASE R18B_step_1 OF
		0:
			//idle
		1:
			TON_62.IN := FALSE;
			EDTPIT0804_record[0] := REAL_TO_INT(EDTPIT0804_PARA.upper_range * 100);
			EDTPIT0804_record[1] := REAL_TO_INT(EDTPIT0804_PARA.upper_range * 100);
			EDTPIT0804_record[2] := REAL_TO_INT(EDTPIT0804_PARA.upper_range * 100);
			EDTTIT0802_record[0] := REAL_TO_INT(EDTTIT0802_PARA.upper_range * 100);
			EDTTIT0802_record[1] := REAL_TO_INT(EDTTIT0802_PARA.upper_range * 100);
			EDTTIT0802_record[2] := REAL_TO_INT(EDTTIT0802_PARA.upper_range * 100);
			R18B_step_1 := 2;
		2:
			EDTTV0802E.input.auto_open_signal := TRUE;
			TON_62.PT := DINT_TO_TIME(EDTP3S1_PARA_T4 * 1000);
			TON_62.IN := TRUE;
			IF TON_62.Q THEN
				TON_62.IN := FALSE;
				R18B_step_1 := 3;
			END_IF;
		3:
			EDTTV0802E.input.auto_open_signal := FALSE;
			EDTTV0802D.input.auto_open_signal := FALSE;
			R18B_step_1 := 4;
		4:
			EDTTV0802A.input.auto_open_signal := TRUE;
			IF EDTTV0802A.input.open_feedback_state THEN
				EDTTV0802B.input.auto_open_signal := TRUE;
			END_IF;
			IF EDTTV0802B.input.open_feedback_state AND EDTTV0802A.input.open_feedback_state THEN
				R18B_step_1 := 5;
			END_IF;
		5:
			//每两秒采集一个数据，连续采集3个，连续下降则判定为温度开始下降
			IF temp_decrease_0802 THEN
				R18B_step_1 := 6;
			END_IF;
		6:
			EDTTV0802B.input.auto_open_signal := FALSE;
			IF EDTTV0802B.input.close_feedback_state THEN
				EDTTV0802A.input.auto_open_signal := FALSE;
			END_IF;
			IF EDTTV0802A.input.close_feedback_state AND EDTTV0802B.input.close_feedback_state THEN
				R18B_step_1 := 7;
			END_IF;
		7:
			EDTTV0802E.input.auto_open_signal := TRUE;
			IF EDTTV0802E.input.open_feedback_state THEN
				EDTXV0813.input.auto_open_signal := TRUE;
				R18B_step_1 := 8;
			END_IF;
		8:
			TON_62.PT := DINT_TO_TIME(EDTP3S1_PARA_T2 * 1000);
			TON_62.IN := TRUE;
			IF TON_62.Q THEN
				TON_62.IN := FALSE;
				R18B_step_1 := 9;
			END_IF;
		9:
			//每两秒采集一个数据，连续采集3个，连续下降则判定值开始下降
			TON_62.PT := DINT_TO_TIME(EDTP3S1_PARA_T1 * 1000);
			TON_62.IN := TRUE;
			IF TON_62.Q THEN
				TON_62.IN := FALSE;
				EDTPIT0804_record[offset_b] := REAL_TO_INT(EDTPIT0804.status.value * 100);
				offset_b := offset_b + 1;
			END_IF;
			IF offset_b > 2 THEN
				offset_b := 0;
			END_IF;
			IF (EDTPIT0804_record[0] > EDTPIT0804_record[1]) AND (EDTPIT0804_record[1] > EDTPIT0804_record[2]) THEN
				R18B_step_1 := 10;
			END_IF;
		10:
			IF EDTPIT0804.status.value <= EDTP3S1_PARA_P3 THEN
				EDTXV0813.input.auto_open_signal := FALSE;
				temp_h_flag_b := FALSE;
				R18B_step_1 := 0;
			END_IF;
	END_CASE;
	TON_62();

	//压力上限
	CASE R18B_step_2 OF
		0:
			//idle
		1:
			EDTPIT0804_record[0] := REAL_TO_INT(EDTPIT0804_PARA.upper_range * 100);
			EDTPIT0804_record[1] := REAL_TO_INT(EDTPIT0804_PARA.upper_range * 100);
			EDTPIT0804_record[2] := REAL_TO_INT(EDTPIT0804_PARA.upper_range * 100);
			TON_65.IN := FALSE;
			EDTTV0802E.input.auto_open_signal := FALSE;
			EDTTV0802D.input.auto_open_signal := FALSE;
			IF EDTTV0802E.input.close_feedback_state AND EDTTV0802D.input.close_feedback_state AND EDTTV0802C.input.close_feedback_state THEN
				R18B_step_2 := 2;
			END_IF;
		2:
			EDTTV0802A.input.auto_open_signal := TRUE;
			IF EDTTV0802A.input.open_feedback_state THEN
				EDTTV0802B.input.auto_open_signal := TRUE;
			END_IF;
			IF EDTTV0802B.input.open_feedback_state AND EDTTV0802A.input.open_feedback_state THEN
				R18B_step_2 := 3;
			END_IF;
		3:
			IF EDTPIT0802.status.value <= EDTP3S1_PARA_P2 THEN
				R18B_step_2 := 4;
			END_IF;
		4:
			EDTTV0802B.input.auto_open_signal := FALSE;
			IF EDTTV0802B.input.close_feedback_state THEN
				EDTTV0802A.input.auto_open_signal := FALSE;
			END_IF;
			IF EDTTV0802A.input.close_feedback_state AND EDTTV0802B.input.close_feedback_state THEN
				R18B_step_2 := 5;
			END_IF;
		5:
			EDTTV0802E.input.auto_open_signal := TRUE;
			IF EDTTV0802E.input.open_feedback_state THEN
				EDTXV0813.input.auto_open_signal := TRUE;
				R18B_step_2 := 6;
			END_IF;
		6:
			TON_65.PT := DINT_TO_TIME(EDTP3S1_PARA_T2 * 1000);
			TON_65.IN := TRUE;
			IF TON_65.Q THEN
				TON_65.IN := FALSE;
				R18B_step_2 := 7;
			END_IF;
		7:
			//每两秒采集一个数据，连续采集3个，连续下降则判定值开始下降
			TON_65.PT := DINT_TO_TIME(EDTP3S1_PARA_T1 * 1000);
			TON_65.IN := TRUE;
			IF TON_65.Q THEN
				TON_65.IN := FALSE;
				EDTPIT0804_record[offset_b] := REAL_TO_INT(EDTPIT0804.status.value * 100);
				offset_b := offset_b + 1;
			END_IF;
			IF offset_b > 2 THEN
				offset_b := 0;
			END_IF;
			IF (EDTPIT0804_record[0] > EDTPIT0804_record[1]) AND (EDTPIT0804_record[1] > EDTPIT0804_record[2]) THEN
				R18B_step_2 := 8;
			END_IF;
		8:
			IF EDTPIT0804.status.value <= EDTP3S1_PARA_P3 THEN
				EDTXV0813.input.auto_open_signal := FALSE;
				press_h_flag_b := FALSE;
				R18B_step_2 := 0;
			END_IF;
	END_CASE;
	TON_65();

	//温度低限
	CASE R18B_step_3 OF
		0:
			//idle
		1:
			EDTTV0802E.input.auto_open_signal := FALSE;
			EDTXV0813.input.auto_open_signal := FALSE;
			EDTTV0802C.input.auto_open_signal := TRUE;
			EDTTV0802D.input.auto_open_signal := TRUE;
			R18B_step_3 := 2;
		2:
			IF EDTTIT0802.status.value >= EDTP3S1_PARA_Temp1 THEN
				R18B_step_3 := 3;
			END_IF;
		3:
			EDTTV0802C.input.auto_open_signal := FALSE;
			EDTTV0802D.input.auto_open_signal := FALSE;
			EDTTV0802E.input.auto_open_signal := TRUE;
			R18B_step_3 := 4;
		4:
			temp_l_flag_b := FALSE;
			R18B_step_3 := 0;
	END_CASE;

	//=======================================================================================================
	//pid 温度调节
	R_TRIG_3(CLK := EDTTVT0802.status.auto_mode);
	IF R_TRIG_3.Q THEN
		MTBasicsPID_7.Enable := TRUE;
	END_IF;
	F_TRIG_3(CLK := EDTTVT0802.status.auto_mode);
	IF F_TRIG_3.Q THEN
		MTBasicsPID_7.Enable := FALSE;
	END_IF;

	//MTBasicsPID_7.Enable := TRUE;
	//MTBasicsPID_7.Invert := TRUE;
	MTBasicsPID_7.PIDParameters.Gain := EDTPid0802Para.gain;
	MTBasicsPID_7.PIDParameters.IntegrationTime := EDTPid0802Para.integration_time;
	MTBasicsPID_7.PIDParameters.DerivativeTime := EDTPid0802Para.derivative_time;
	MTBasicsPID_7.MinOut := 0.0;
	MTBasicsPID_7.MaxOut := 100.0;
	MTBasicsPID_7.SetValue := EDTPid0802Para.set_value;
	MTBasicsPID_7.ActValue := EDTTIT0802.status.value;
	MTBasicsPID_7.Update := EDTPid0802.update;
	MTBasicsPID_7();
	EDTPid0802.out := MTBasicsPID_7.Out;
	IF MTBasicsPID_7.Active THEN
		EDTTVT0802.input.auto_degree_set := MTBasicsPID_7.Out;
	ELSE
		EDTTVT0802.input.auto_degree_set := 0.0;
	END_IF;
	IF MTBasicsPID_7.UpdateDone THEN
		EDTPid0802.update := FALSE;
	END_IF;

	//人工确认步骤可用
	IF (EDTP3S1B.status.run_state) AND (NOT EDTP3S1B_STEP[EDTP3S1B.status.run_step].done AND ((EDTP3S1B.status.run_step = 3))) THEN
		EDTP3S1B.status.confirm_enable := TRUE;
	ELSE
		EDTP3S1B.status.confirm_enable := FALSE;
	END_IF;
END_ACTION
